// TwinCAT 3 PLC project fms205plc
// ProgramVersion: 3.1.4023.0
// libraries:
//   CmpBitmapPool, * (System)
//   Tc2_Standard, * (Beckhoff Automation GmbH)
//   Tc2_System, * (Beckhoff Automation GmbH)
//   Tc3_Module, * (Beckhoff Automation GmbH)
//   VisuDialogs, * (System)
//   VisuSymbols,3.5.10.0,System
// project tree:
//   / GlobalTextList.TcGTLO, PlcTask.TcTTO (not stored), Visualization Manager.TcVMO (not stored)
//   L1 Architecture/ L1_ModuleBase.TcPOU, L1_Actuator.TcPOU, L1_ControllerBase_SFC.TcPOU, L1_Director.TcPOU, L1_GEMMA.TcDUT, L1_Sensor.TcPOU
//   L2 Module Controllers/ L2_Alimentador_SFC.TcPOU, L2_Cinta_SFC.TcPOU, L2_Evacuador_SFC.TcPOU, L2_MedidorTapa_SFC.TcPOU, L2_PickAndPlace_SFC.TcPOU, L2_PlatoDivisor_SFC.TcPOU, L2_Simple_SFC.TcPOU
//   L3 Modules/ L3_Alimentador.TcPOU, L3_CaptadorInductivo.TcPOU, L3_Cinta.TcPOU, L3_DetectorFotoelectrico.TcPOU, L3_Evacuador.TcPOU, L3_MedidorTapa.TcPOU, L3_PickAndPlace.TcPOU, L3_PlatoDivisor.TcPOU
//   L4 Station Controllers/ L4_FMS205_F1Producir_SFC.TcPOU, L4_FMS205_F2SeqPrep_SFC.TcPOU, L4_FMS205_F3SeqFin_SFC.TcPOU, L4_FMS205_F6Prueba_SFC.TcPOU
//   L5 Station User Interfaces/ L5_Constantes.TcGVL, L5_Panel.TcPOU, L5_FMS205VISU.TcVIS, L5_ImagePool.TcIPO (not stored)
//   L6 Station/ L6_FMS205.TcPOU, L6_Tapas.TcPOU, MAIN.TcPOU
// real-time tasks:
//   TASK PlcTask: cycle T#10ms, priority 20, ADS port 350
// I/O:
//   DEVICE Dispositivo 1 (EtherCAT) (disabled), AmsNetId 192.168.1.58.2.1
//     Terminal 1 (EK1200) [EK1200-5000 EtherCAT Power supply (2A E-Bus)]
//       Terminal 2 (EL1008) [EL1008 8Ch. Dig. Input 24V, 3ms]
//       Terminal 3 (EL1008) [EL1008 8Ch. Dig. Input 24V, 3ms]
//       Terminal 4 (EL2008) [EL2008 8Ch. Dig. Output 24V, 0.5A]
//       Terminal 5 (EL2008) [EL2008 8Ch. Dig. Output 24V, 0.5A]
//       Terminal 6 (EL1008) [EL1008 8Ch. Dig. Input 24V, 3ms]
//       Terminal 7 (EL1008) [EL1008 8Ch. Dig. Input 24V, 3ms]
//       Terminal 8 (EL2008) [EL2008 8Ch. Dig. Output 24V, 0.5A]
//       Terminal 9 (EL2008) [EL2008 8Ch. Dig. Output 24V, 0.5A]
//       Terminal 10 (EL5151) [EL5151 1Ch. Inc. Encoder]
//       Terminal 11 (EL9011) [EL9011 End Terminal]
// variable links:
//   fms205plc/fms205plc Instance <-> Device 1 (EtherCAT)/Term 1 (EK1200)/Term 10 (EL5151)
//     PlcTask Inputs/MAIN.fbFMS205.mdMedidorTapa.dh <-> ENC Inputs/dh
//   fms205plc/fms205plc Instance <-> Device 1 (EtherCAT)/Term 1 (EK1200)/Term 2 (EL1008)
//     PlcTask Inputs/MAIN.fbFMS205.fbPanel.hwPE_Seta <-> Channel 1/PE
//     PlcTask Inputs/MAIN.fbFMS205.fbPanel.hwPM_PulsadorMarcha <-> Channel 3/PM
//     PlcTask Inputs/MAIN.fbFMS205.fbPanel.hwPOC_PulsadorReset <-> Channel 5/POC
//     PlcTask Inputs/MAIN.fbFMS205.fbPanel.hwPS_PulsadorStop <-> Channel 4/PS
//     PlcTask Inputs/MAIN.fbFMS205.fbPanel.hwSM_SelecAutoManual <-> Channel 2/SM
//     PlcTask Inputs/MAIN.fbFMS205.mdCinta.cp0.hwValue <-> Channel 7/cp0
//     PlcTask Inputs/MAIN.fbFMS205.mdCinta.cp1.hwValue <-> Channel 8/cp1
//     PlcTask Inputs/MAIN.fbFMS205.mdCinta.pp.hwValue <-> Channel 6/pp
//   fms205plc/fms205plc Instance <-> Device 1 (EtherCAT)/Term 1 (EK1200)/Term 3 (EL1008)
//     PlcTask Inputs/MAIN.fbFMS205.mdCinta.cp2.hwValue <-> Channel 1/cp2
//   fms205plc/fms205plc Instance <-> Device 1 (EtherCAT)/Term 1 (EK1200)/Term 4 (EL2008)
//     PlcTask Outputs/MAIN.fbFMS205.fbPanel.hwLA_LamparaAlarma <-> Channel 2/LA
//     PlcTask Outputs/MAIN.fbFMS205.fbPanel.hwLM_LamparaMarcha <-> Channel 3/LM
//     PlcTask Outputs/MAIN.fbFMS205.mdAlimentador.FM.hwValue <-> Channel 4/FM
//     PlcTask Outputs/MAIN.fbFMS205.mdCinta.REV.hwValue <-> Channel 6/REV
//     PlcTask Outputs/MAIN.fbFMS205.mdCinta.RUN.hwValue <-> Channel 5/RUN
//     PlcTask Outputs/MAIN.fbFMS205.mdCinta.R_1.hwValue <-> Channel 7/R+
//     PlcTask Outputs/MAIN.fbFMS205.mdCinta.S_1.hwValue <-> Channel 8/S+
//   fms205plc/fms205plc Instance <-> Device 1 (EtherCAT)/Term 1 (EK1200)/Term 5 (EL2008)
//     PlcTask Outputs/MAIN.fbFMS205.fbPanel.hwAS_AvisadorSonoro <-> Channel 1/AS
//   fms205plc/fms205plc Instance <-> Device 1 (EtherCAT)/Term 1 (EK1200)/Term 6 (EL1008)
//     PlcTask Inputs/MAIN.fbFMS205.mdEvacuador.f0.hwValue <-> Channel 6/f0
//     PlcTask Inputs/MAIN.fbFMS205.mdEvacuador.f1.hwValue <-> Channel 7/f1
//     PlcTask Inputs/MAIN.fbFMS205.mdEvacuador.g0.hwValue <-> Channel 8/g0
//     PlcTask Inputs/MAIN.fbFMS205.mdPickAndPlaceCarga.h0.hwValue <-> Channel 1/a0
//     PlcTask Inputs/MAIN.fbFMS205.mdPickAndPlaceCarga.h1.hwValue <-> Channel 2/a1
//     PlcTask Inputs/MAIN.fbFMS205.mdPickAndPlaceCarga.v0.hwValue <-> Channel 3/b0
//     PlcTask Inputs/MAIN.fbFMS205.mdPickAndPlaceCarga.v1.hwValue <-> Channel 4/b1
//     PlcTask Inputs/MAIN.fbFMS205.mdPlatoDivisor.d0.hwValue <-> Channel 5/d0
//   fms205plc/fms205plc Instance <-> Device 1 (EtherCAT)/Term 1 (EK1200)/Term 7 (EL1008)
//     PlcTask Inputs/MAIN.fbFMS205.mdAlimentador.k1.hwValue <-> Channel 6/k1
//     PlcTask Inputs/MAIN.fbFMS205.mdCaptadorInductivo.di.hwValue <-> Channel 7/di
//     PlcTask Inputs/MAIN.fbFMS205.mdDetectorFotoelectrico.df.hwValue <-> Channel 8/df
//     PlcTask Inputs/MAIN.fbFMS205.mdEvacuador.v1.hwValue <-> Channel 1/v1
//     PlcTask Inputs/MAIN.fbFMS205.mdPickAndPlaceDescarga.h0.hwValue <-> Channel 2/h0
//     PlcTask Inputs/MAIN.fbFMS205.mdPickAndPlaceDescarga.h1.hwValue <-> Channel 3/h1
//     PlcTask Inputs/MAIN.fbFMS205.mdPickAndPlaceDescarga.v0.hwValue <-> Channel 4/i0
//     PlcTask Inputs/MAIN.fbFMS205.mdPickAndPlaceDescarga.v1.hwValue <-> Channel 5/i1
//   fms205plc/fms205plc Instance <-> Device 1 (EtherCAT)/Term 1 (EK1200)/Term 8 (EL2008)
//     PlcTask Outputs/MAIN.fbFMS205.mdEvacuador.F_0.hwValue <-> Channel 7/F-
//     PlcTask Outputs/MAIN.fbFMS205.mdEvacuador.F_1.hwValue <-> Channel 6/F+
//     PlcTask Outputs/MAIN.fbFMS205.mdEvacuador.G_1.hwValue <-> Channel 8/G+
//     PlcTask Outputs/MAIN.fbFMS205.mdPickAndPlaceCarga.HOR.hwValue <-> Channel 1/A+
//     PlcTask Outputs/MAIN.fbFMS205.mdPickAndPlaceCarga.PIN.hwValue <-> Channel 3/C+
//     PlcTask Outputs/MAIN.fbFMS205.mdPickAndPlaceCarga.VER.hwValue <-> Channel 2/B+
//     PlcTask Outputs/MAIN.fbFMS205.mdPlatoDivisor.D_1.hwValue <-> Channel 4/D+
//     PlcTask Outputs/MAIN.fbFMS205.mdPlatoDivisor.E_1.hwValue <-> Channel 5/E+
//   fms205plc/fms205plc Instance <-> Device 1 (EtherCAT)/Term 1 (EK1200)/Term 9 (EL2008)
//     PlcTask Outputs/MAIN.fbFMS205.mdAlimentador.K_1.hwValue <-> Channel 5/K+
//     PlcTask Outputs/MAIN.fbFMS205.mdEvacuador.V_1.hwValue <-> Channel 1/V+
//     PlcTask Outputs/MAIN.fbFMS205.mdMedidorTapa.L_1.hwValue <-> Channel 6/L+
//     PlcTask Outputs/MAIN.fbFMS205.mdPickAndPlaceDescarga.HOR.hwValue <-> Channel 2/H+
//     PlcTask Outputs/MAIN.fbFMS205.mdPickAndPlaceDescarga.PIN.hwValue <-> Channel 4/J+
//     PlcTask Outputs/MAIN.fbFMS205.mdPickAndPlaceDescarga.VER.hwValue <-> Channel 3/I+

// ---- L1 Architecture/L1_GEMMA.TcDUT
{attribute 'qualified_only'}
{attribute 'strict'}
TYPE L1_GEMMA :
(
	  (* Modos de la Guia de Estudio de los Modos de Marcha y Parada *)
    (* [Modes du Guide d'Etude des Modes de Marche et d'Arrêt] *)
    (* [Modes of Study Guide of the Modes of Operating and Stopping] *)

    (* Procedimientos de parada [les procédures d'arrets/stop procedures] *)
    A1ParadaInicial, (*  0: parada en el estado inicial
               [arrêt dans etat initial] 
               [stopped in the initial state] *)
    A2ParaFinCiclo, (*  1: parada solicitada a final de ciclo
               [arret demandé en fin de cycle] 
               [requested end cycle stop] *)
    A3ParadaEstado, (*  2: parada solicitada en un estado determinado
               [arret demande dans etat determine] 
               [requested particular state stop] *)
    A4ParadaObtenida, (*  3: parada obtenida
               [arret obtenu] 
               [obteined stop] *)
    A5PreparandoTrasFallo, (*  4: preparacion para la recuperacion del fallo
               [preparation pour remise en route apres defaillance] 
               [preparation for the recovery of the failure] *)
    A6Inicializando, (*  5: situando la PO en el estado inicial
               [mise PO dans état initial] 
               [set the PO in initial state] *)
    A7SituandoEstado, (*  6: situando la PO en un estado determinado
               [mise PO dans état déterminé]
               [set the PO in a certain state] *)

    (* Procedimientos de funcionamiento [les procédures de fonctionnement/operating procedures] *)
    F1ProduccionNormal, (*  7: produccion normal
               [production normale] 
               [normal operation] *)
    F2SecuenciaPreparacion, (*  8: secuencia de preparacion
               [marche de preparation] 
               [preparation sequence] *)
    F3SecuenciaFinalizacion, (*  9: secuencia de finalizacion
               [marche de cloture] 
               [ending sequence] *)
    F4VerificacionSinOrden, (* 10: verificacion en desorden
               [marche de verification dans le desordre] 
               [verification with no order] *)
    F5VerificacionOrdenada, (* 11: verificacion en orden
               [marche de verification dans l'ordre] 
               [verification whit order] *)
    F6Probando, (* 12: prueba
               [marche de test] 
               [test] *)

    (* Procedimientos de fallo [les procédures en défaillances] *)
    D1ParadaEmergencia, (* 13: parada de emergencia
               [arret d'urgence] 
               [emergency stop] *)
    D2TratamientoFallos, (* 14: diagnostico y/o tratamiento de los fallos
               [diagnostic et/ou traitement de la défaillance] 
               [diagnosis and/or treatment of failures] *)
    D3ProducirConFallos  (* 15: produccion a pesar de los fallos
               [production tout de même] 
               [production despite the failures] *)
);
END_TYPE

// ---- L5 Station User Interfaces/L5_Constantes.TcGVL
// {attribute 'qualified_only'}
VAR_GLOBAL CONSTANT
	clModeAFill : DWORD := 16#FF808080;;
	clModeFFill : DWORD := 16#FFFF0000;
	clModeDFill : DWORD := 16#FF800000;
	
	colDesFill		 : DWORD :=16#FFFF0000;	
	colDesFont		 : DWORD :=16#FFFFFFFF;	
	colDesFrameSin	 : DWORD :=16#FFFF0000;		
	colVacFill		 : DWORD :=16#FFF2F2F2;	
	colVacFont		 : DWORD :=16#FF000000;	
	colVacFrameSin	 : DWORD :=16#FFF2F2F2;		
	colTapFill		 : DWORD :=16#FFFFFF00;	
	colTapFont		 : DWORD :=16#FF000000;	
	colTapFrameSin	 : DWORD :=16#FF000000;		
	colClaFill		 : DWORD :=16#FFFFFF00;	
	colClaFont		 : DWORD :=16#FF000000;	
	colClaFrameSin	 : DWORD :=16#FF000000;		
	colOscFill		 : DWORD :=16#FFFFFF00;	
	colOscFont		 : DWORD :=16#FF000000;	
	colOscFrameSin	 : DWORD :=16#FF000000;		
	colAluFill		 : DWORD :=16#FF808080;	
	colAluFont		 : DWORD :=16#FFFFFFFF;	
	colAluFrameSin	 : DWORD :=16#FF000000;	
	colAluFrameOk	 : DWORD :=16#FF00B050;	
	colAluFrameKo	 : DWORD :=16#FFFF0000;
	colBlnFill		 : DWORD :=16#FFFFFFFF;	
	colBlnFont		 : DWORD :=16#FF000000;	
	colBlnFrameSin	 : DWORD :=16#FF000000;	
	colBlnFrameOk	 : DWORD :=16#FF00B050;	
	colBlnFrameKo	 : DWORD :=16#FFFF0000;
	colNgrFill		 : DWORD :=16#FF0D0D0D;	
	colNgrFont		 : DWORD :=16#FFFFFFFF;	
	colNgrFrameSin	 : DWORD :=16#FF000000;	
	colNgrFrameOk	 : DWORD :=16#FF00B050;	
	colNgrFrameKo	 : DWORD :=16#FFFF0000;
	colErrFill		 : DWORD :=16#FFFF0000;	
	colErrFont		 : DWORD :=16#FFFFFFFF;	
	colErrFrameSin	 : DWORD :=16#FF000000;		

	// aparte el grosor de la línea debe establecerse a 3
	colModFillExec	 : DWORD :=16#50FFFF00; // amarillo
	colModFramExec	 : DWORD :=16#FFFFA500; // naranja
	colModFillDone	 : DWORD :=16#5000C000; // verde
	colModFramDone	 : DWORD :=16#FF004000; // verde oscuro
	colModFillReady	 : DWORD :=16#00FFFF00; // amarillo transparente
	colModFramReady	 : DWORD :=16#00FFA500; // naranja transparente
	
	// Posiciones
	MoverMax		: REAL := -1.0;
	MaxAlimeY		: REAL := 100;
	MaxCargaX		: REAL := 80;
	MaxDescaY		: REAL := 90;
	MinCintaX		: REAL := -200;
	MaxCintaX		: REAL := 145;
	
	MaxPosDesca		: REAL := 100;	// mismo valor que deja el brazo de descarga	
	MaxPosEvacu		: REAL := 100;
	MinPosCarro		: REAL := -200;
	MaxPosCarro		: REAL := 145;


END_VAR

// ---- L1 Architecture/L1_ModuleBase.TcPOU
FUNCTION_BLOCK L1_ModuleBase

VAR_INPUT
	dr		: REFERENCE TO L1_Director;
	ID		: BYTE; 		// identificador de la unidad funcional (el módulo)
	Name	: STRING;		// Nombre del módulo (para erroers)
	Execute	: BOOL;
	Ack		: BOOL;
END_VAR

VAR_OUTPUT
	IC			: BOOL;
	Ready		: BOOL;
	Failure		: BOOL;
	FailName 	: STRING;
	Done		: BOOL;
END_VAR

END_FUNCTION_BLOCK

// ---- L1 Architecture/L1_Director.TcPOU
FUNCTION_BLOCK L1_Director
(*

Módulo L1_Director

Entrada: consignas generadas a partir del panel físico, la interfaz de usuario y el estado de la estación
Salida: nuevo estado de Gemma

1. Consignas

	cnA2_FinCiclo:			Solicitud de que la estación se detenga cuando acabe el ciclo
	cnA3_Estado:			Solicitud de que la estación se detenga lo antes posible
	cnA6_Inicializar: 		Solicitud de inicialización de la estación
	
	cnF0_Empezar: 			Solicitud de empezar a Producir/Pobar o continuar después de una parada/fallo
	cnF1_Producir:			Solicitud de producción, incluyendo secuencias de preparación=F2/finalización=F3
	cnF2_Preparar:			Solicitud de que la estación ejecute la secuencia de praparación antes de empezar el lote
	cnF3_Finalizar:			Solicitud de que se ejecute la secuencia de finalización después de acabar el lote
	cnF4_Planta:			Solicitud de paso al modo manual
	cnF5_Funcion:			Solicitud de prueba de grafcets a nivel de módulo
	cnF6_Probar				Solicitud de prueba secuencial de la estación (monolítico)

	cnD1_Emergencia: 		Solicitud de parada de emergencia


2. Estado de la estación

	IC:						La estación cumple las condiciones iniciales
	Failure:				Alguno de los módulos de la estación ha fallado
	EndCycle:				La estación ha terminado un ciclo de producción
	EndBatch:				La estación ha terminado de producir el lote
	IsPaused:				Todos los módulos de la estación se han detenido

3. Modos GEMMA
	A1ParadaInicial:		La estación está parada esperando instrucciones
	A2ParaFinCiclo:			Estación produciendo pero se detendrá cuando se termine el ciclo actual
	A3ParadaEstado:			Estación en marcha pero se detendrá en cuanto alcance un estado estable (IsSafe)
	A4ParadaObtenida: 		La estación está detenida después de alcanzar un estado estable
	A5PreparandoTrasFallo:	La estación está cambiando al modo anterior a que se produjera el fallo
	A6Inicializadndo:		Estación inicializando esperando a que se cumplan las condiciones iniciales
	A7SituandoEstado:		Modo no tratado 
	
	F1ProduccionNormal:		Estación produciendo el lote piezas
	F2SecuenciaPreparacion:	Estación preparándose para producir (evaluando qué hay en cada sector del plato)
	F3SecuenciaFinalizacion:Estación finalizando la producción (vaciando las tapas que quedan en el plato)	
	F4VerificacionSinOrden:	Estación en modo manual
	F5VerificacionOrdenada: Estación ejecutando un Grafcet a nivel de módulo
	F6Probando:				Estación ejecutando el Grafcet secuencial (monolítico)

	D1ParadaEmergencia: 	Estación ha entrado en parada de emergencia
	D2TratamientoFallos:	Estación detenida (o en modo F4) para corregir el fallo que se ha producido
	D3ProducirConFallos:	Estado no tratado

	
*)

VAR CONSTANT
	gmColorArret 	: DWORD := 16#FF808080;
	gmColorFonct 	: DWORD := 16#FF000080;
	gmColorDefail 	: DWORD := 16#FF800000;
END_VAR

VAR_INPUT
	IC 				: BOOL := TRUE; 			// todos los módulos están en condiciones iniciales
	IsPaused		: BOOL := TRUE; 			// estación en estado estable con todos los módulos detenidos
	EndCycle		: BOOL := FALSE;			// se ha completado un ciclo con/sin rechazo/descarga
	EndBatch		: BOOL := FALSE; 			// se han completado todas las tapas del lote
	Failure			: BOOL := FALSE;			// hay al menos un módulo que ha fallado

	cnA1_ParadaIni	: BOOL;
	cnF0_Empezar	: BOOL;
	
	
	cnF1_Producir	: BOOL;
	cnF2_Preparar	: BOOL;
	//IsPrepared		: BOOL := TRUE; 			// secuencia de preparación completada
	
	cnA2_FinCiclo	: BOOL;
	cnA3_Estado		: BOOL;
	cnF3_Finalizar	: BOOL;
	//IsFinished		: BOOL := TRUE; 			// secuencia de finalización completada
	
	cnF5_Funcion	: BOOL; 					// modo verificación ordenada
	cnF6_Probar		: BOOL;

	cnF4_Planta		: BOOL; 					// modo verificación sin orden	
	cnD1_Emergencia	: BOOL; 					// pulsar la seta
	cnA6_Inicializar: BOOL;
	//cnF1_Reanudar	: BOOL;

END_VAR

VAR_OUTPUT
	gmLocalHost		: BOOL 		:= FALSE; 		// TODO - SUSTITUIR ESTO POR LA CONDICIÓN DE LOCALHOST		
	gmModeActual	: L1_GEMMA 	:= L1_GEMMA.A6Inicializando; 		// Modo GEMMA actual
	gmModePrev		: L1_GEMMA; 				// Modo GEMMA anterior al actual
	gmModeColor		: DWORD 	:= gmColorArret;
	Tic				: BOOL		:= FALSE; 		// Se activa y desactiva cada 500 ms
	Clock			: TON;						// Temporizador para activar/desactivar Tic
END_VAR	

VAR
	gmFamiArret		: BOOL 		:= TRUE; 		// Familia de parada
	gmFamiFonct		: BOOL 		:= FALSE; 		// Familia de funcionamiento
	gmFamiDefail	: BOOL 		:= FALSE; 		// Familia de salida de fallos
	
	Speed			: REAL := 100.0;			// Velocidad variable de los controladores
	LastSpeed		: real := 0;			// para calcular sólo si hay cambio de velocidad
	
	
	//---------------------------------- dt_ Defalut Times	
	dt_MaximoTiempoRespuesta	: TIME := T#5S;				// Tiempos generales
	dt_TiempoReinicio			: TIME := T#5S;	
	dt_K_1 						: TIME := T#1S;				// Temporizador empujador tapa
	dt_R_1						: TIME := T#0.5S;			// Temporizador retenedor de la cinta
	dt_S_1						: TIME := T#0.5S;			// Temporizador separador de la cinta
	dt_EP						: TIME := T#0.5S;			// Tiempo de entrada del pale
	dt_TP						: TIME := T#1S;				// Tiempo de transferencia del pale
	dt_XP						: TIME := T#1S;				// Tiempo de salida del pale
	dt_SOL 						: TIME := T#100MS; 			// tiempo después de soltar y antes de subir
	dt_V_1						: TIME := T#5S;				// tiempo máximo succionando sin que se active el sensor v1
	dt_L_1						: TIME := T#1S;				// tiempo máximo de bajada del medidor de tapas
	dt_PIN 						: TIME := T#1S;				// tiempo para pinzar una tapa antes de subir el brazo
	dt_E_1						: TIME := T#400MS;			// tiempo para que el retenedor bloquee el plato
	dt_D_1 						: TIME := T#1.4S;			// tiempo para girar el plato a la siguiente posición
END_VAR


VAR_OUTPUT
	tmMaximoTiempoRespuesta		: TIME := dt_MaximoTiempoRespuesta;
	tmTiempoReinicio			: TIME := dt_TiempoReinicio;	
	tmK_1 						: TIME := dt_K_1;			// Temporizador empujador tapa
	tmR_1						: TIME := dt_R_1;			// Temporizador retenedor de la cinta
	tmS_1						: TIME := dt_S_1;			// Temporizador separador de la cinta
	tmEP						: TIME := dt_EP;			// Tiempo de entrada del pale
	tmTP						: TIME := dt_TP;			// Tiempo de transferencia del pale
	tmXP						: TIME := dt_XP;			// Tiempo de salida del pale
	tmSOL 						: TIME := dt_SOL; 			// tiempo después de soltar y antes de subir
	tmV_1						: TIME := dt_V_1;			// tiempo máximo succionando sin que se active el sensor v1
	tmL_1						: TIME := dt_L_1;		// tiempo máximo de bajada del medidor de tapas
	tmPIN 						: TIME := dt_PIN;		// tiempo para pinzar una tapa antes de subir el brazo
	tmE_1						: TIME := dt_E_1;		// tiempo para que el retenedor bloquee el plato
	tmD_1 						: TIME := dt_D_1;		// tiempo para girar el plato a la siguiente posición
END_VAR

METHOD ProcessCycle : BOOL
// Actualiza el reloj y la veloidad cada medio segundo
Clock(IN := NOT Clock.Q, PT:=T#500MS);
IF Clock.Q THEN
	Tic := NOT Tic;
	UpdateSpeed();
END_IF


IF cnD1_Emergencia AND NOT cnF4_Planta THEN
    gmModeActual 		:= L1_GEMMA.D1ParadaEmergencia;
//	gmModePrev 			:= L1_GEMMA.D1ParadaEmergencia;
//	IF cnF4_Planta THEN 				
//		gmModePrev := L1_GEMMA.D1ParadaEmergencia
//		gmModeActual := L1_GEMMA.F4VerificacionSinOrden;
//	ELSE
//		; // desde emergencia se puede pasar a F4 (desarmando la seta)				
//	END_IF
//		
	
ELSIF cnA6_Inicializar and not cnF4_Planta THEN 
    gmModeActual 		:= L1_GEMMA.A6Inicializando;
	// gmModePrev 			:= L1_GEMMA.L1_GEMMA.A6Inicializando;	

END_IF
	
    CASE gmModeActual OF
		
	
        (* ------------------------------------------------------------ Procedimientos de parada *)
		
        L1_GEMMA.A6Inicializando: (* A6 -> A1 o F4 *)
			gmModePrev := L1_GEMMA.A6Inicializando;
            IF IC THEN 
                gmModeActual := L1_GEMMA.A1ParadaInicial;
			ELSIF cnF4_Planta THEN 				
                gmModeActual := L1_GEMMA.F4VerificacionSinOrden;
            END_IF

			
			
			
        L1_GEMMA.A1ParadaInicial: (* A1 -> A6, F4, F5, F2 o F6 *)
			gmModePrev := L1_GEMMA.A1ParadaInicial;
            IF NOT IC THEN // IF NOT Restaurada THEN
                gmModeActual := L1_GEMMA.A6Inicializando;				
            ELSIF cnF4_Planta THEN 				
                gmModeActual := L1_GEMMA.F4VerificacionSinOrden;				
			ELSIF cnF5_Funcion THEN 
				gmModeActual := L1_GEMMA.F5VerificacionOrdenada;             
			ELSIF cnF1_Producir AND cnF0_Empezar THEN
                gmModeActual := L1_GEMMA.F2SecuenciaPreparacion;
			ELSIF cnF6_Probar AND cnF0_Empezar THEN
				gmModeActual := L1_GEMMA.F6Probando;
			ELSE
				; // Esperar a que se pulse el bortón de marcha
            END_IF

			
			
        L1_GEMMA.F4VerificacionSinOrden: (* F4 -> ModePrev *)
            //IF Failure THEN
			//	gmModeActual := L1_GEMMA.D2TratamientoFallos;				
            //ELSIF NOT cnF4_Planta THEN
			IF NOT cnF4_Planta THEN 				
				gmModeActual := gmModePrev; // al salir del modo planta volver al modo previo				
            ELSE                
                ; // Seguir en modo manual
            END_IF

			
			
		L1_GEMMA.F1ProduccionNormal, 		
        L1_GEMMA.A2ParaFinCiclo,
        L1_GEMMA.F2SecuenciaPreparacion, 	
		L1_GEMMA.F3SecuenciaFinalizacion, 	
        L1_GEMMA.F5VerificacionOrdenada,  	
		L1_GEMMA.F6Probando: 				        
			// retorno desde tratamiento de errores y planta
			IF gmModeActual=L1_GEMMA.F5VerificacionOrdenada THEN
				gmModePrev := L1_GEMMA.A1ParadaInicial; 								// F5 retorna a A1
			ELSE
				gmModePrev := gmModeActual;												// Resto retorna donde quedó			
			END_IF			
			
			// cambios de modo actual
            IF Failure THEN 															// cualquiera -> D2
                gmModeActual := L1_GEMMA.D2TratamientoFallos;
            ELSIF cnA3_Estado THEN				
				gmModeActual := L1_GEMMA.A3ParadaEstado; 								// cualquiera -> A3
			ELSIF cnF4_Planta THEN 				
                gmModeActual := L1_GEMMA.F4VerificacionSinOrden;						// cualquiera -> F4
            ELSIF gmModeActual=L1_GEMMA.F2SecuenciaPreparacion AND NOT cnF2_Preparar THEN 	// F2-> F1
                gmModeActual:= L1_GEMMA.F1ProduccionNormal;
			ELSIF gmModeActual=L1_GEMMA.F1ProduccionNormal AND cnA2_FinCiclo THEN 		// F1 -> A2				
				gmModeActual:= L1_GEMMA.A2ParaFinCiclo;
			ELSIF gmModeActual=L1_GEMMA.A2ParaFinCiclo AND EndCycle THEN 				// A2 -> A3
				gmModePrev  := L1_GEMMA.F1ProduccionNormal; 							// A2 -> A3 ... -> F1
                gmModeActual:= L1_GEMMA.A3ParadaEstado;
			ELSIF gmModeActual=L1_GEMMA.F1ProduccionNormal AND EndBatch THEN 			// F1-> F3
                gmModeActual:= L1_GEMMA.F3SecuenciaFinalizacion;
			ELSIF gmModeActual=L1_GEMMA.F3SecuenciaFinalizacion AND NOT cnF3_Finalizar THEN // F3 -> A1
				gmModeActual:= L1_GEMMA.A1ParadaInicial;
			ELSIF gmModeActual=L1_GEMMA.F5VerificacionOrdenada AND NOT cnF5_Funcion THEN // F5 -> A1
				gmModeActual:= L1_GEMMA.A1ParadaInicial;				
			ELSIF gmModeActual=L1_GEMMA.F6Probando AND NOT cnF6_Probar THEN 			// F6 -> A1
				gmModeActual:= L1_GEMMA.A1ParadaInicial; 
            ELSE                
                ; // continuar con la preparación/producción/finalización
            END_IF
			

			
        L1_GEMMA.A3ParadaEstado: 
			IF Failure THEN																// A3 -> D2
                gmModeActual := L1_GEMMA.D2TratamientoFallos;
			ELSIF IsPaused THEN															// A3 -> A4
                gmModeActual := L1_GEMMA.A4ParadaObtenida;
            ELSE
                ; // Seguir produciendo hasta que todos los módulos paren en un estado estable
            END_IF
            			
        L1_GEMMA.A4ParadaObtenida:
			IF cnF0_Empezar THEN														// A4 -> retorna
				gmModeActual := gmModePrev; // retomar el estado antes de la parada
			ELSE
				; // seguir parada hasta la consigna de reanudar	
			END_IF
                    
		L1_GEMMA.A5PreparandoTrasFallo:
			gmModeActual := gmModePrev;		// Volver al estado anterior al fallo 
			
        L1_GEMMA.A7SituandoEstado: (* Situando la PO en un estado determinado *)
            ; // estado no tratado en la FMS205

			
			
        (* ------------------------------------------------------------ Procedimientos de funcionamiento *)
        
			
			
			
			
        	
			
        (* ------------------------------------------------------------ Procedimientos de defecto *)
        L1_GEMMA.D1ParadaEmergencia: (* Parada de emergencia *)
			IF NOT cnD1_Emergencia THEN //  TODO CONSIGNA DE EMERGENCIA DEBE TENER ENCUENTA LA POC
                gmModeActual := L1_GEMMA.A6Inicializando; // Al quitar la parada de emergencia hay que reinicializar la estación
			ELSIF cnF4_Planta then							// desde A1 se puede entrar F4 para arreglar el problema
				gmModePrev := L1_GEMMA.D1ParadaEmergencia;
				gmModeActual := L1_GEMMA.F4VerificacionSinOrden;
            ELSE                
                ; // Esperar a que se quite la parada de emergencia
            END_IF
			
        L1_GEMMA.D2TratamientoFallos: (* Diagnostico/tratamiento de los fallos *)
            IF NOT Failure THEN // el fallo se resuelve por sí solo (no debería pasar)
                gmModeActual := L1_GEMMA.A5PreparandoTrasFallo;
			ELSIF cnF4_Planta THEN // se pasa a modo F4 para arreglarlo
				gmModeActual := L1_GEMMA.F4VerificacionSinOrden;
            ELSIF cnF0_Empezar THEN // se pulsa Marcha para intentar recuperar                
                gmModeActual := L1_GEMMA.A5PreparandoTrasFallo;
            END_IF

        L1_GEMMA.D3ProducirConFallos: (* Produccion a pesar de los fallos *)
            ; // estado no tratado en la FMS205

    END_CASE
// END_IF

(* PARAMETROS DE SALIDA *)
gmFamiArret  := (gmModeActual >= L1_GEMMA.A1ParadaInicial) AND (gmModeActual <= L1_GEMMA.A7SituandoEstado);
gmFamiFonct  := (gmModeActual >= L1_GEMMA.F1ProduccionNormal) AND (gmModeActual <= L1_GEMMA.F6Probando);
gmFamiDefail := (gmModeActual >= L1_GEMMA.D1ParadaEmergencia) AND (gmModeActual <= L1_GEMMA.D3ProducirConFallos);
gmModeColor := SEL(gmFamiArret,SEL(gmFamiFonct, gmColorDefail, gmColorFonct), gmColorArret);

UpdateSpeed();
//UpdateUi(pn:=pn);
END_METHOD

METHOD UpdateSpeed : BOOL

VAR
	factor : REAL;
END_VAR
IF Speed <= 0 THEN
	Speed := 1;
ELSIF Speed<>LastSpeed THEN
	LastSpeed := Speed; // sólo se ejecuta el código la primera vez que cambia la velocidad
	
	factor := 100.0/Speed;
	
	tmMaximoTiempoRespuesta		:= TO_TIME(TO_REAL(dt_MaximoTiempoRespuesta) * factor);
	tmTiempoReinicio			:= TO_TIME(TO_REAL(dt_TiempoReinicio) * factor);
	tmK_1 						:= TO_TIME(TO_REAL(dt_K_1) * factor);					// Temporizador empujador tapa
	tmR_1						:= TO_TIME(TO_REAL(dt_R_1) * factor);					// Temporizador retenedor de la cinta
	tmS_1						:= TO_TIME(TO_REAL(dt_S_1) * factor);					// Temporizador separador de la cinta
	tmEP						:= TO_TIME(TO_REAL(dt_EP) * factor);					// Tiempo de entrada del pale
	tmTP						:= TO_TIME(TO_REAL(dt_TP) * factor);					// Tiempo de transferencia del pale
	tmXP						:= TO_TIME(TO_REAL(dt_XP) * factor);					// Tiempo de salida del pale
	tmSOL 						:= TO_TIME(TO_REAL(dt_SOL) * factor); 					// tiempo después de soltar y antes de subir
	tmV_1						:= TO_TIME(TO_REAL(dt_V_1) * factor);					// tiempo máximo succionando sin que se active el sensor v1
	tmL_1						:= TO_TIME(TO_REAL(dt_L_1) * factor);					// tiempo máximo de bajada del medidor de tapas
	tmPIN 						:= TO_TIME(TO_REAL(dt_PIN) * factor);					// tiempo para pinzar una tapa antes de subir el brazo
	tmE_1						:= TO_TIME(TO_REAL(dt_E_1) * factor);					// tiempo para que el retenedor bloquee el plato
	tmD_1 						:= TO_TIME(TO_REAL(dt_D_1) * factor);					// tiempo para girar el plato a la siguiente posición
	
END_IF
END_METHOD

END_FUNCTION_BLOCK

// ---- L1 Architecture/L1_Actuator.TcPOU
FUNCTION_BLOCK L1_Actuator

VAR CONSTANT
END_VAR

VAR_OUTPUT
	uiValue			: BOOL;					// Vinculación a la visualización
	uiToolTip		: STRING;				// Tooltip en la visualización
END_VAR

VAR
	hwValue AT %Q*	: BOOL;					// Vinculación al hardware de la estación	
END_VAR

METHOD ForceValue : BOOL
VAR_INPUT
	NewValue : BOOL;
END_VAR
uiValue := NewValue;
hwValue := NewValue;
END_METHOD

METHOD ProcessCycle : BOOL
VAR_INPUT
	gmMode		: L1_GEMMA;
	sfcValue 	: BOOL;		// estado del actuador devuelto por el Grafcet
END_VAR
IF gmMode = L1_GEMMA.F4VerificacionSinOrden THEN	
	hwValue := uiValue;	// Actualizar el hardware con la entrada desde la visualización
ELSE	
	hwValue := sfcValue; // Actualizar el hardware y la visualicación con la entrada desde el Grafcet
	uiValue := sfcValue;
END_IF
END_METHOD

END_FUNCTION_BLOCK

// ---- L1 Architecture/L1_ControllerBase_SFC.TcPOU
FUNCTION_BLOCK L1_ControllerBase_SFC

VAR_INPUT
	dr			: REFERENCE TO L1_Director;		// acceso a todos los tiempos de espera
	IC			: BOOL;
	Execute		: BOOL;
	Ack			: BOOL;	
	SFCPause	: BOOL;
	SFCReset	: BOOL;
	UnsafeStop 	: BOOL;
	Clocks		: ARRAY[1..MAX_ERRORS]	OF TON; 
END_VAR

VAR_OUTPUT
	Ready		: BOOL;
	Executing	: BOOL;
	_Performed	: BOOL;					// Para poner la primera vez que se leen los sensores o se gira el plato
	Done		: BOOL := FALSE;
	Timed		: ARRAY[1..MAX_ERRORS]	OF BOOL; 
	NumError	: UINT := 0;
	gmModePrev	: L1_GEMMA := L1_GEMMA.A6Inicializando;	
	colPicFill	: DWORD; // color para destacar en la foto según esté Ready (tranparente), Ejecutando (amarillo) o Esperando Ack (verde) 
	colPicFram	: DWORD; // color del marco  	
END_VAR

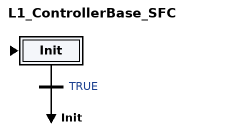
INITIAL_STEP Init:
END_STEP
TRANSITION FROM Init TO Init
    := TRUE;
END_TRANSITION

METHOD FB_init : BOOL

VAR_INPUT
	bInitRetains : BOOL; // if TRUE, the retain variables are initialized (warm start / cold start)
	bInCopyCode : BOOL;  // if TRUE, the instance afterwards gets moved into the copy code (online change)
END_VAR

VAR 
	I: UINT;
END_VAR
NumError		:= 0;					// Inicializar el estado a 0 (no hay error)
_Performed		:= FALSE;
UnsafeStop 		:= FALSE;
Done			:= FALSE;
gmModePrev		:= L1_GEMMA.A6Inicializando;

FOR I:=1 TO MAX_ERRORS DO				// Inicializar todos los flags de etapas temporizadas
	Timed[i] 		:= FALSE;
END_FOR
END_METHOD

METHOD IsPaused : BOOL
IsPaused := SFCPause;
END_METHOD

PROPERTY Performed : BOOL
GET
Performed := _Performed;
END_GET
SET
_Performed := Performed;
END_SET
END_PROPERTY

METHOD ProcessCycle : BOOL

VAR_INPUT
	gmMode : L1_GEMMA;
END_VAR

VAR 
	i : UINT;
END_VAR
// Tratamiento del reset
IF gmModePrev<>gmMode AND gmMode=L1_GEMMA.A6Inicializando THEN
	gmModePrev	:= gmMode;
	SFCReset 	:= TRUE;
	Ready		:= FALSE; 
	Executing	:= FALSE;
	_Performed	:= FALSE;				// Para poner la primera vez que se leen los sensores o se gira el plato
	Done		:= FALSE;
	NumError	:= 0;
	colPicFill	:= colModFillReady;  
	colPicFram	:= colModFramReady;   	
ELSE
	SFCReset 	:= FALSE;
END_IF
gmModePrev := gmMode;

// Tratamiento de la parada
SFCPause := NOT UnsafeStop AND (NumError <> 0 
	OR gmMode=L1_GEMMA.A3ParadaEstado OR gmMode=L1_GEMMA.A4ParadaObtenida or gmMode=L1_GEMMA.D1ParadaEmergencia);

// Tratamiento de errores
FOR i:= 1 TO MAX_ERRORS DO			
	Clocks[i](IN:= Timed[i], PT:=MAX_TIMEOUT);
	IF Clocks[i].Q THEN								// si saltó algún temporizador, devolver su número como error
		NumError := i;
		EXIT;
	END_IF
END_FOR


// Tratamiento del color en la foto
IF Ready THEN
	Executing 	:= FALSE;
	Performed 	:= FALSE;
	colPicFill	:= colModFillReady;
	colPicFram	:= colModFramReady;
ELSIF Done THEN
	Executing 	:= FALSE;
	colPicFill	:= colModFillDone;
	colPicFram	:= colModFramDone;	
ELSE
	Executing 	:= TRUE;
	colPicFill	:= colModFillExec;
	colPicFram	:= colModFramExec;	
END_IF
END_METHOD

METHOD ResetError : BOOL
NumError := 0;
END_METHOD

END_FUNCTION_BLOCK

// ---- L1 Architecture/L1_Sensor.TcPOU
FUNCTION_BLOCK L1_Sensor

VAR_OUTPUT
	uiValue			: BOOL;					
END_VAR

VAR	
	hwValue AT %I*	: BOOL;					// Vinculación al hardware de la estación
	uiToolTip		: STRING;				// Tooltip en la visualización
END_VAR

METHOD ProcessCycle : BOOL
VAR_INPUT
	LocalHost	: BOOL;
END_VAR
VAR_OUTPUT
	sfcValue 	: BOOL;		// estado del sensor que se entregará al Grafcet
END_VAR
IF LocalHost THEN	
	hwValue := uiValue; 	// simulando la estación, el valor del sensor depende de la interfaz	
ELSE	
	uiValue := hwValue; 	// ejecutando en la estación, el valor de la visualización depende del hardware
END_IF
sfcValue := hwValue;		// estado del sensor que se entregará al Grafcet
END_METHOD

END_FUNCTION_BLOCK

// ---- L2 Module Controllers/L2_Alimentador_SFC.TcPOU
FUNCTION_BLOCK L2_Alimentador_SFC EXTENDS L1_ControllerBase_SFC

VAR_INPUT 					// Sensores y comandos
	k1	: BOOL; 			// Sensor de empujador tapa delante
	Alimentar :BOOL;
END_VAR

VAR_OUTPUT					// Actuadores
	Leyendo: BOOL;	
	K_1: BOOL; 				// Actuador de empujador tapa avanza	 
	FM : BOOL; 
END_VAR

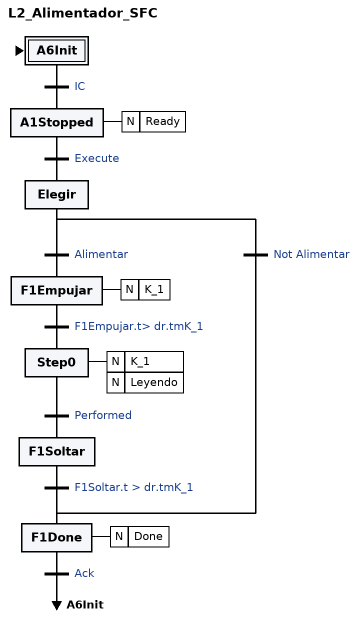
INITIAL_STEP A6Init:
END_STEP
TRANSITION FROM A6Init TO A1Stopped
    := IC;
END_TRANSITION
STEP A1Stopped:
    Ready(N);
END_STEP
TRANSITION FROM A1Stopped TO Elegir
    := Execute;
END_TRANSITION
STEP Elegir:
END_STEP
TRANSITION FROM Elegir TO F1Empujar
    := Alimentar;
END_TRANSITION
STEP F1Empujar:
    K_1(N);
END_STEP
TRANSITION FROM F1Empujar TO Step0
    := F1Empujar.t> dr.tmK_1;
END_TRANSITION
STEP Step0:
    K_1(N);
    Leyendo(N);
END_STEP
TRANSITION FROM Step0 TO F1Soltar
    := Performed;
END_TRANSITION
STEP F1Soltar:
END_STEP
TRANSITION FROM F1Soltar TO F1Done
    := F1Soltar.t > dr.tmK_1;
END_TRANSITION
TRANSITION FROM Elegir TO F1Done
    := Not Alimentar;
END_TRANSITION
STEP F1Done:
    Done(N);
END_STEP
TRANSITION FROM F1Done TO A6Init
    := Ack;
END_TRANSITION

END_FUNCTION_BLOCK

// ---- L2 Module Controllers/L2_Cinta_SFC.TcPOU
FUNCTION_BLOCK L2_Cinta_SFC  EXTENDS L1_ControllerBase_SFC

VAR_INPUT 					// Sensores y comandos
	Situar		: BOOL;
	Transferir	: BOOL;	
	pp			: BOOL; 	// presencia de pale
	cp0			: BOOL;
	cp1			: BOOL;
	cp2			: BOOL;
END_VAR

VAR_OUTPUT					// Actuadores
	RUN			: BOOL; 	// activa motor
	REV			: BOOL; 	// invierte motor
	R_1			: BOOL; 	// retenedor baja
	S_1			: BOOL; 	// separador sube
END_VAR

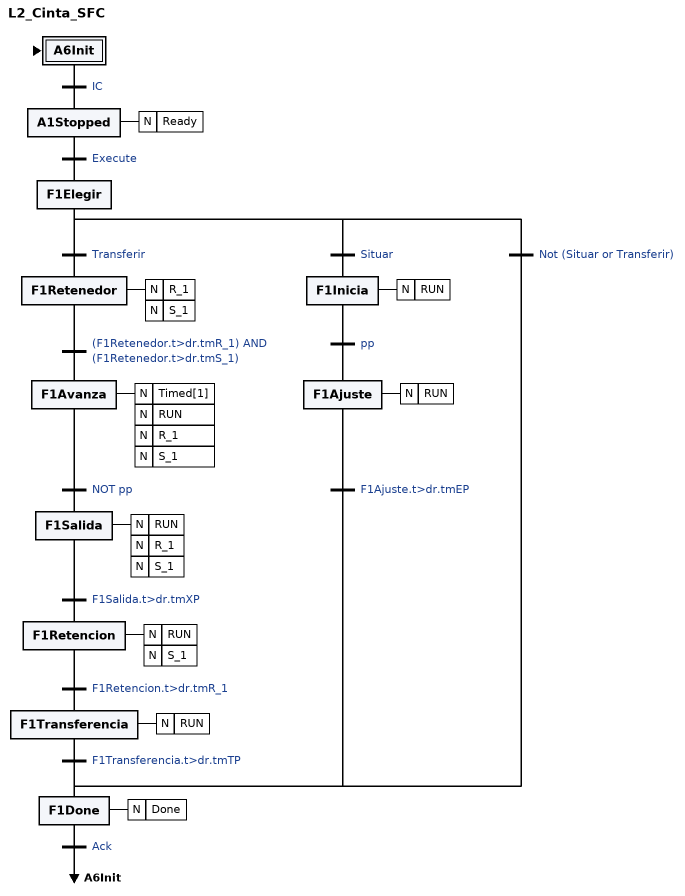
INITIAL_STEP A6Init:
END_STEP
TRANSITION FROM A6Init TO A1Stopped
    := IC;
END_TRANSITION
STEP A1Stopped:
    Ready(N);
END_STEP
TRANSITION FROM A1Stopped TO F1Elegir
    := Execute;
END_TRANSITION
STEP F1Elegir:
END_STEP
TRANSITION FROM F1Elegir TO F1Retenedor
    := Transferir;
END_TRANSITION
STEP F1Retenedor:
    R_1(N);
    S_1(N);
END_STEP
TRANSITION FROM F1Retenedor TO F1Avanza
    := (F1Retenedor.t>dr.tmR_1) AND (F1Retenedor.t>dr.tmS_1);
END_TRANSITION
STEP F1Avanza:
    Timed[1](N);
    RUN(N);
    R_1(N);
    S_1(N);
END_STEP
TRANSITION FROM F1Avanza TO F1Salida
    := NOT pp;
END_TRANSITION
STEP F1Salida:
    RUN(N);
    R_1(N);
    S_1(N);
END_STEP
TRANSITION FROM F1Salida TO F1Retencion
    := F1Salida.t>dr.tmXP;
END_TRANSITION
STEP F1Retencion:
    RUN(N);
    S_1(N);
END_STEP
TRANSITION FROM F1Retencion TO F1Transferencia
    := F1Retencion.t>dr.tmR_1;
END_TRANSITION
STEP F1Transferencia:
    RUN(N);
END_STEP
TRANSITION FROM F1Transferencia TO F1Done
    := F1Transferencia.t>dr.tmTP;
END_TRANSITION
TRANSITION FROM F1Elegir TO F1Inicia
    := Situar;
END_TRANSITION
STEP F1Inicia:
    RUN(N);
END_STEP
TRANSITION FROM F1Inicia TO F1Ajuste
    := pp;
END_TRANSITION
STEP F1Ajuste:
    RUN(N);
END_STEP
TRANSITION FROM F1Ajuste TO F1Done
    := F1Ajuste.t>dr.tmEP;
END_TRANSITION
TRANSITION FROM F1Elegir TO F1Done
    := Not (Situar or Transferir);
END_TRANSITION
STEP F1Done:
    Done(N);
END_STEP
TRANSITION FROM F1Done TO A6Init
    := Ack;
END_TRANSITION

END_FUNCTION_BLOCK

// ---- L2 Module Controllers/L2_Evacuador_SFC.TcPOU
FUNCTION_BLOCK L2_Evacuador_SFC EXTENDS L1_ControllerBase_SFC

VAR_INPUT 				// Sensores y comandos
	Evacuar		: BOOL; // Hay que evacuar la tapa en la posición del módulo
	f0        	: BOOL; (* gh0 (nombre=f0  c=I22 B=J2 b=22 módulo=EL1008 T=6  C=6 etiqueta=-B10, input) Pick and place de rechazo detrás *)
    f1        	: BOOL; (* gh1 (nombre=f1  c=I23 B=J2 b=06 módulo=EL1008 T=6  C=6 etiqueta=-B11, input) Pick and place de rechazo delante *)
    g0        	: BOOL; (* gv1 (nombre=g0  c=I24 B=J2 b=31 módulo=EL1008 T=6  C=6 etiqueta=-B12, input) Pick and place de rechazo arriba *)
    v1        	: BOOL; (* ge1 (nombre=v1  c=I25 B=J1 b=25 módulo=EL1008 T=7  C=7 etiqueta=-B13, input) Pick and place de rechazo vacío *)
END_VAR

VAR_OUTPUT				// Actuadores
	F_1       	: BOOL; (* gHRA (nombre=F+  c=Q22 B=J2  b=35 módulo=EL2008 T=8 C=8 etiqueta=-Y8,  output) Pick and place de rechazo avanza (afuera) *)
    F_0       	: BOOL; (* gHRR (nombre=F-  c=Q23 B=J2  b=32 módulo=EL2008 T=8 C=8 etiqueta=-Y9,  output) Pick and place de rechazo retrocede *)
    G_1       	: BOOL; (* gVER (nombre=G+  c=Q24 B=J2  b=11 módulo=EL2008 T=8 C=8 etiqueta=-Y10, output) Pick and place de rechazo baja *)
    V_1       	: BOOL; (* gEYE (nombre=V+  c=Q25 B=J2  b=08 módulo=EL2008 T=9 C=9 etiqueta=-Y11, output) Pick and place de rechazo succiona *)
END_VAR

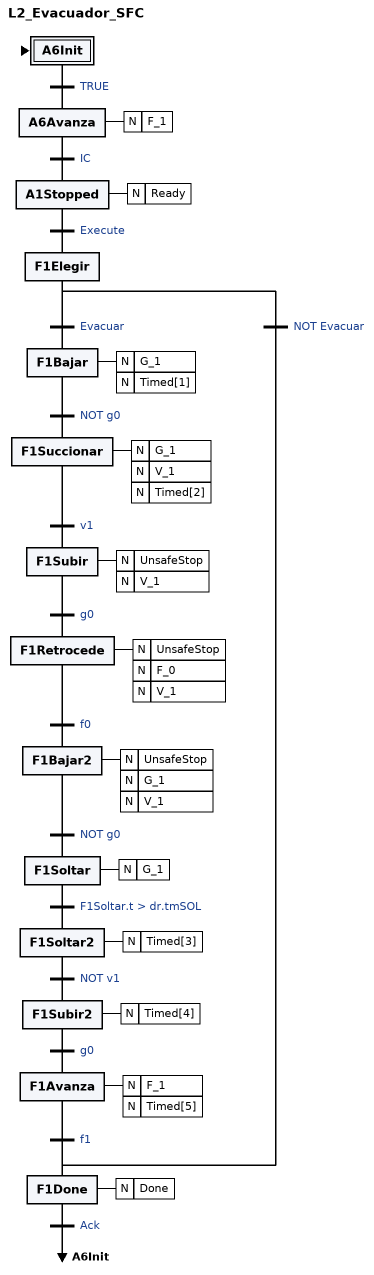
INITIAL_STEP A6Init:
END_STEP
TRANSITION FROM A6Init TO A6Avanza
    := TRUE;
END_TRANSITION
STEP A6Avanza:
    F_1(N);
END_STEP
TRANSITION FROM A6Avanza TO A1Stopped
    := IC;
END_TRANSITION
STEP A1Stopped:
    Ready(N);
END_STEP
TRANSITION FROM A1Stopped TO F1Elegir
    := Execute;
END_TRANSITION
STEP F1Elegir:
END_STEP
TRANSITION FROM F1Elegir TO F1Bajar
    := Evacuar;
END_TRANSITION
STEP F1Bajar:
    G_1(N);
    Timed[1](N);
END_STEP
TRANSITION FROM F1Bajar TO F1Succionar
    := NOT g0;
END_TRANSITION
STEP F1Succionar:
    G_1(N);
    V_1(N);
    Timed[2](N);
END_STEP
TRANSITION FROM F1Succionar TO F1Subir
    := v1;
END_TRANSITION
STEP F1Subir:
    UnsafeStop(N);
    V_1(N);
END_STEP
TRANSITION FROM F1Subir TO F1Retrocede
    := g0;
END_TRANSITION
STEP F1Retrocede:
    UnsafeStop(N);
    F_0(N);
    V_1(N);
END_STEP
TRANSITION FROM F1Retrocede TO F1Bajar2
    := f0;
END_TRANSITION
STEP F1Bajar2:
    UnsafeStop(N);
    G_1(N);
    V_1(N);
END_STEP
TRANSITION FROM F1Bajar2 TO F1Soltar
    := NOT g0;
END_TRANSITION
STEP F1Soltar:
    G_1(N);
END_STEP
TRANSITION FROM F1Soltar TO F1Soltar2
    := F1Soltar.t > dr.tmSOL;
END_TRANSITION
STEP F1Soltar2:
    Timed[3](N);
END_STEP
TRANSITION FROM F1Soltar2 TO F1Subir2
    := NOT v1;
END_TRANSITION
STEP F1Subir2:
    Timed[4](N);
END_STEP
TRANSITION FROM F1Subir2 TO F1Avanza
    := g0;
END_TRANSITION
STEP F1Avanza:
    F_1(N);
    Timed[5](N);
END_STEP
TRANSITION FROM F1Avanza TO F1Done
    := f1;
END_TRANSITION
TRANSITION FROM F1Elegir TO F1Done
    := NOT Evacuar;
END_TRANSITION
STEP F1Done:
    Done(N);
END_STEP
TRANSITION FROM F1Done TO A6Init
    := Ack;
END_TRANSITION

END_FUNCTION_BLOCK

// ---- L2 Module Controllers/L2_MedidorTapa_SFC.TcPOU
FUNCTION_BLOCK L2_MedidorTapa_SFC EXTENDS L1_ControllerBase_SFC

VAR_INPUT 							// Sensores y comandos
	dh					: UINT; 	// Detector valor altura 
	Medir				: BOOL; // Lectura_Registrada	: BOOL;		// La lectura de la altura ha terminado 	
END_VAR

VAR_OUTPUT							// Actuadores
	L_1: BOOL; 						// Medidor de altura baja
	Leyendo: BOOL;
END_VAR

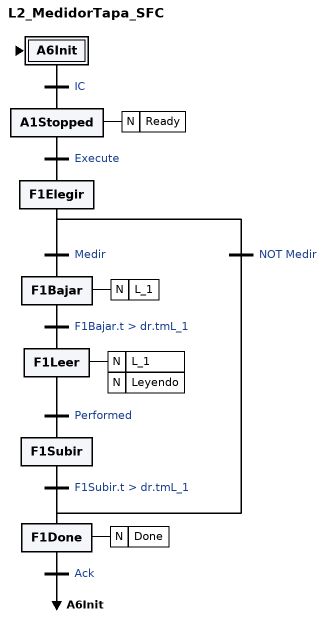
INITIAL_STEP A6Init:
END_STEP
TRANSITION FROM A6Init TO A1Stopped
    := IC;
END_TRANSITION
STEP A1Stopped:
    Ready(N);
END_STEP
TRANSITION FROM A1Stopped TO F1Elegir
    := Execute;
END_TRANSITION
STEP F1Elegir:
END_STEP
TRANSITION FROM F1Elegir TO F1Bajar
    := Medir;
END_TRANSITION
STEP F1Bajar:
    L_1(N);
END_STEP
TRANSITION FROM F1Bajar TO F1Leer
    := F1Bajar.t > dr.tmL_1;
END_TRANSITION
STEP F1Leer:
    L_1(N);
    Leyendo(N);
END_STEP
TRANSITION FROM F1Leer TO F1Subir
    := Performed;
END_TRANSITION
STEP F1Subir:
END_STEP
TRANSITION FROM F1Subir TO F1Done
    := F1Subir.t > dr.tmL_1;
END_TRANSITION
TRANSITION FROM F1Elegir TO F1Done
    := NOT Medir;
END_TRANSITION
STEP F1Done:
    Done(N);
END_STEP
TRANSITION FROM F1Done TO A6Init
    := Ack;
END_TRANSITION

END_FUNCTION_BLOCK

// ---- L2 Module Controllers/L2_PickAndPlace_SFC.TcPOU
FUNCTION_BLOCK L2_PickAndPlace_SFC EXTENDS L1_ControllerBase_SFC

VAR_INPUT 				// Sensores y comandos
	h0		: BOOL; 	(* Final de carrera horizontal retraida *)
	h1		: BOOL; 	(* Final de carrera horizontal extendido *)
	v1		: BOOL; 	(*Final de carrera vertical abajo*)
	v0		: BOOL; 	(*Final de carrera vertical arriba*)
	Mover	: BOOL;
END_VAR

VAR_OUTPUT			// Actuadores
	HOR		: BOOL; (* Actuador de extension de brazo horizontal *)
	VER		: BOOL; (* Actuador de movimiento vertical de brazo*)
	PIN		: BOOL; (*Actuador de pinza de brazo*)
END_VAR

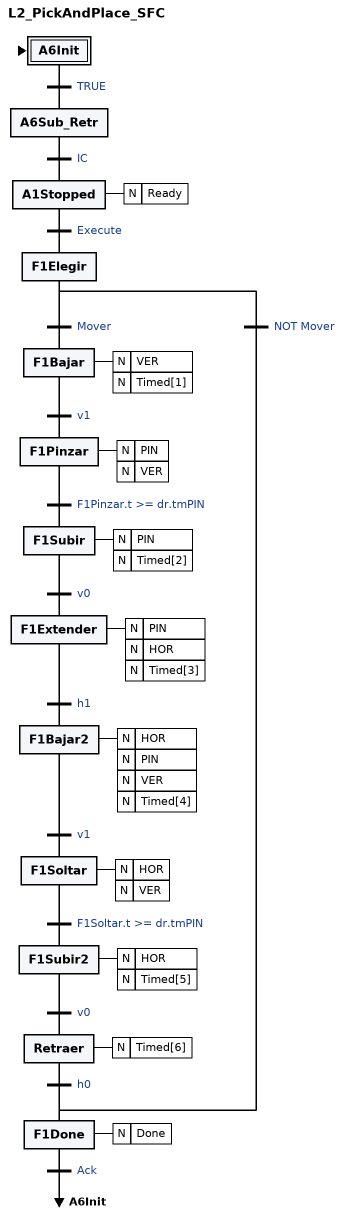
INITIAL_STEP A6Init:
END_STEP
TRANSITION FROM A6Init TO A6Sub_Retr
    := TRUE;
END_TRANSITION
STEP A6Sub_Retr:
END_STEP
TRANSITION FROM A6Sub_Retr TO A1Stopped
    := IC;
END_TRANSITION
STEP A1Stopped:
    Ready(N);
END_STEP
TRANSITION FROM A1Stopped TO F1Elegir
    := Execute;
END_TRANSITION
STEP F1Elegir:
END_STEP
TRANSITION FROM F1Elegir TO F1Bajar
    := Mover;
END_TRANSITION
STEP F1Bajar:
    VER(N);
    Timed[1](N);
END_STEP
TRANSITION FROM F1Bajar TO F1Pinzar
    := v1;
END_TRANSITION
STEP F1Pinzar:
    PIN(N);
    VER(N);
END_STEP
TRANSITION FROM F1Pinzar TO F1Subir
    := F1Pinzar.t >= dr.tmPIN;
END_TRANSITION
STEP F1Subir:
    PIN(N);
    Timed[2](N);
END_STEP
TRANSITION FROM F1Subir TO F1Extender
    := v0;
END_TRANSITION
STEP F1Extender:
    PIN(N);
    HOR(N);
    Timed[3](N);
END_STEP
TRANSITION FROM F1Extender TO F1Bajar2
    := h1;
END_TRANSITION
STEP F1Bajar2:
    HOR(N);
    PIN(N);
    VER(N);
    Timed[4](N);
END_STEP
TRANSITION FROM F1Bajar2 TO F1Soltar
    := v1;
END_TRANSITION
STEP F1Soltar:
    HOR(N);
    VER(N);
END_STEP
TRANSITION FROM F1Soltar TO F1Subir2
    := F1Soltar.t >= dr.tmPIN;
END_TRANSITION
STEP F1Subir2:
    HOR(N);
    Timed[5](N);
END_STEP
TRANSITION FROM F1Subir2 TO Retraer
    := v0;
END_TRANSITION
STEP Retraer:
    Timed[6](N);
END_STEP
TRANSITION FROM Retraer TO F1Done
    := h0;
END_TRANSITION
TRANSITION FROM F1Elegir TO F1Done
    := NOT Mover;
END_TRANSITION
STEP F1Done:
    Done(N);
END_STEP
TRANSITION FROM F1Done TO A6Init
    := Ack;
END_TRANSITION

END_FUNCTION_BLOCK

// ---- L2 Module Controllers/L2_PlatoDivisor_SFC.TcPOU
FUNCTION_BLOCK L2_PlatoDivisor_SFC EXTENDS L1_ControllerBase_SFC

VAR_INPUT 					// Sensores y comandos
	d0  		: BOOL; 
END_VAR

VAR_OUTPUT					// Actuadores
	D_1 		: BOOL; 
    E_1 		: BOOL; 
END_VAR

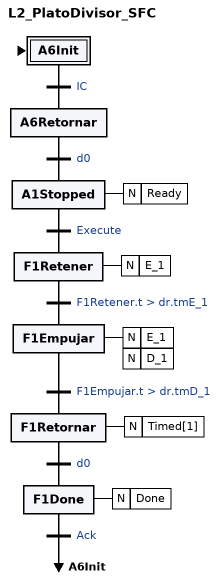
INITIAL_STEP A6Init:
END_STEP
TRANSITION FROM A6Init TO A6Retornar
    := IC;
END_TRANSITION
STEP A6Retornar:
END_STEP
TRANSITION FROM A6Retornar TO A1Stopped
    := d0;
END_TRANSITION
STEP A1Stopped:
    Ready(N);
END_STEP
TRANSITION FROM A1Stopped TO F1Retener
    := Execute;
END_TRANSITION
STEP F1Retener:
    E_1(N);
END_STEP
TRANSITION FROM F1Retener TO F1Empujar
    := F1Retener.t > dr.tmE_1;
END_TRANSITION
STEP F1Empujar:
    E_1(N);
    D_1(N);
END_STEP
TRANSITION FROM F1Empujar TO F1Retornar
    := F1Empujar.t > dr.tmD_1;
END_TRANSITION
STEP F1Retornar:
    Timed[1](N);
END_STEP
TRANSITION FROM F1Retornar TO F1Done
    := d0;
END_TRANSITION
STEP F1Done:
    Done(N);
END_STEP
TRANSITION FROM F1Done TO A6Init
    := Ack;
END_TRANSITION

END_FUNCTION_BLOCK

// ---- L2 Module Controllers/L2_Simple_SFC.TcPOU
FUNCTION_BLOCK L2_Simple_SFC EXTENDS L1_ControllerBase_SFC
// Grafcet simple para los detectores fotoeléctrico e inductivo

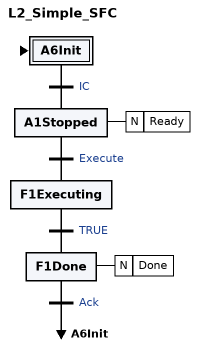
INITIAL_STEP A6Init:
END_STEP
TRANSITION FROM A6Init TO A1Stopped
    := IC;
END_TRANSITION
STEP A1Stopped:
    Ready(N);
END_STEP
TRANSITION FROM A1Stopped TO F1Executing
    := Execute;
END_TRANSITION
STEP F1Executing:
END_STEP
TRANSITION FROM F1Executing TO F1Done
    := TRUE;
END_TRANSITION
STEP F1Done:
    Done(N);
END_STEP
TRANSITION FROM F1Done TO A6Init
    := Ack;
END_TRANSITION

END_FUNCTION_BLOCK

// ---- L3 Modules/L3_Alimentador.TcPOU
FUNCTION_BLOCK L3_Alimentador EXTENDS L1_ModuleBase
(*  MÓDULO ALIMENTACIÓN - Manual de usuario #31/27

Para el almacenamiento y posterior alimentación de las tapas, se utiliza un 
cargador de gravedad, provisto de un empujador accionado mediante cilindro 
neumático que realiza la extracción  *)
VAR_INPUT
	Alimentar		: BOOL;
END_VAR

VAR_OUTPUT	
	fbController	: L2_Alimentador_SFC:=(dr:=dr);	
	k1 				: L1_Sensor;
	K_1 			: L1_Actuator;
	FM 				: L1_Actuator; 
	//_TapaAlimentada	: BOOL;
	FaltaMaterial	: BOOL;
	// Position		: REAL:= 0;
	Leyendo			: BOOL;
END_VAR

METHOD ProcessCycle : BOOL 
VAR_INPUT	
	dr			: REFERENCE TO L1_Director;
	tapas		: REFERENCE TO L6_Tapas;
		
END_VAR
IF dr.gmModeActual = L1_GEMMA.A6Inicializando THEN
	//_TapaAlimentada 			:= FALSE;
	FaltaMaterial				:= FALSE;
ELSE
	// Sensores y condiciones iniciales
	k1.ProcessCycle(LocalHost:=dr.gmLocalHost, sfcValue=>fbController.k1);
	IC:=TRUE; 

	// Controlador
	fbController.ProcessCycle(dr.gmModeActual);
	fbController(Alimentar:=Alimentar, dr:=dr, IC:=IC, Leyendo=>Leyendo, Execute:=Execute, Ack:=Ack, Ready=>Ready, Done=>Done);
	
	// Actuadores y actualización de tapas
	IF Ready AND NOT tapas.EstaAlimentada THEN // 	TapaAlimentada THEN 
		tapas.MoverAlime(Delta:=0); // 	Position := 0;												// Inicialmente la posición es arriba
	ELSIF fbController.Leyendo AND NOT fbController.Performed THEN
		fbController.Performed	:= TRUE;
		FaltaMaterial			:= k1.uiValue;
		//_TapaAlimentada 		:= NOT FaltaMaterial;
		tapas.EstaAlimentada	:= NOT FaltaMaterial;
	ELSIF Done AND NOT fbController.Performed AND Alimentar THEN
		tapas.MoverAlime(Delta:=MoverMax);// Position				:= MaxPosAlime;						// Posición final junto al brazo de carga 
	ELSIF fbController.Executing AND Alimentar THEN // Position < MaxPosAlime AND 
		tapas.MoverAlime(Delta:=1); // Position := Position + 1;									// animación de tapa moviendo hacia abajo		
	END_IF	
	K_1.ProcessCycle(gmMode:=dr.gmModeActual, sfcValue:=fbController.K_1);
	FM.ProcessCycle (gmMode:=dr.gmModeActual, sfcValue:=FaltaMaterial AND dr.Tic);
END_IF
END_METHOD

END_FUNCTION_BLOCK

// ---- L6 Station/L6_Tapas.TcPOU
FUNCTION_BLOCK L6_Tapas
VAR CONSTANT
	ColSecIndeterm	: DWORD := 16#80101010; // gris claro
	ColSecVacio		: DWORD := 16#80808080; // gris oscuro
	ColSecPendiente : DWORD := 16#80000080; // azul
	ColSecDescargar	: DWORD := 16#80008000; // verde
	ColSecEvacuar	: DWORD := 16#80800000; // rojo
END_VAR

VAR_INPUT
	ReqNumero	: DINT := 5; 		// requisito de número de tapas deseadas
	ReqAlta		: REAL := 18.5;  	// requisito de tapa alta
	ReqVacio	: REAL := 2.0; 		// si mide menos el sector está vacío

	ReqAluBaja	: BOOL := TRUE;
	ReqAluAlta	: BOOL := TRUE;
	ReqBlnBaja  : BOOL := TRUE;
    ReqBlnAlta  : BOOL := TRUE;
	ReqNgrBaja  : BOOL := FALSE;
    ReqNgrAlta  : BOOL := FALSE; 

	ResPend	  	: DINT := 0;
	ResReal		: DINT := 0;
	ResRech   	: DINT := 0;
END_VAR

(*
VAR_OUTPUT
	FaltaMat	: BOOL; 
	ExeAlime	: BOOL;	
	AckAlime	: BOOL;
	ExeCarga	: BOOL;
	AckCarga	: BOOL;
	ExeMedid	: BOOL;
	ExeFotoe	: BOOL;
	ExeInduc	: BOOL;
	ExeEvacu	: BOOL;
	AckEvacu	: BOOL;
	ExeDesca	: BOOL;
	AckDesca	: BOOL;
	ExeDescaAnt	: BOOL;
	ExePlato	: BOOL;
	AckPlato	: BOOL;
	ExeSitua	: BOOL;
	ExeTrans	: BOOL;
END_VAR
*)


VAR
	_AlimeEsta	: BOOL; // Esta alimentada o no
	_CargaEsta	: BOOL;
	_DescaEsta	: BOOL;
	
	AlimeY		: REAL; // posición vertical de la tapa alimentándose
	CargaX		: REAL; 
	DescaX		: REAL:=MaxCintaX;
	DescaY		: REAL:=MaxDescaY;
	CintaX		: REAL:=MaxCintaX;
	
	
	//NumGiros 	: DINT := 0;
	PosCarga	: DINT;
	PosFotoe	: DINT;
	PosMedid	: DINT;
	PosInduc	: DINT;
	PosEvacu	: DINT;
	PosDesca	: DINT;
	Alimentada	: BOOL; // HAY UNA TAPA EN EL ALIMENTADOR ESPERANDO A SER CARGADA

	//angulo	 	: REAL := 0.0;
	//anguloanim 	: REAL := 0.0; // angulo para animación que gira lentamente
	//HaGirado	: BOOL := FALSE;
	//Falta_Material		: BOOL;

	vEvacuar_Tapa		: ARRAY[0..7] OF BOOL;
	vDescargar_Tapa		: ARRAY[0..7] OF BOOL;
	
	vInicializando 		: ARRAY[0..7] OF BOOL;	
	//vCargar_Tapa		: ARRAY[0..7] OF BOOL;
	vTapa_Cargada 		: ARRAY[0..7] OF BOOL;
	vAltura_Medida		: ARRAY[0..7] OF BOOL;
	vAltura_Pulsos 		: ARRAY[0..7] OF DWORD;
	vAltura_Mm 			: ARRAY[0..7] OF REAL;
	vTapa_Alta			: ARRAY[0..7] OF BOOL;
	vClaridad_Medida	: ARRAY[0..7] OF BOOL;
	vTapa_Clara 		: ARRAY[0..7] OF BOOL;	
	vMateral_Medido		: ARRAY[0..7] OF BOOL;	
	vTapa_Metalica 		: ARRAY[0..7] OF BOOL;	
	vstrUi 				: ARRAY[0..7] OF STRING;
	vstrToolTip			: ARRAY[0..7] OF STRING;
	vColorSector		: ARRAY[0..7] OF DWORD;
	
	vColorFill			: ARRAY[0..7] OF DWORD;
	vColorFont			: ARRAY[0..7] OF DWORD;	
	vColorFrame			: ARRAY[0..7] OF DWORD;

	Evacu_strUi			: STRING;
	Evacu_strToolTip	: STRING;	
	Evacu_ColorFont		: DWORD;
	Evacu_ColorFrame	: DWORD;
	Evacu_ColorFill		: DWORD;
	Evacu_PosX			: REAL;
	Evacu_PosY			: REAL;
	
	Desca_strUi			: STRING;
	Desca_strToolTip	: STRING;	
	Desca_ColorFont		: DWORD;
	Desca_ColorFrame	: DWORD;
	Desca_ColorFill		: DWORD;
	Desca_PosX			: REAL;
	Desca_PosY			: REAL;

	
END_VAR

METHOD Actualizar : BOOL
VAR_INPUT
END_VAR

VAR
	i 	: INT := 0;
END_VAR

FOR i:=0 TO 7 DO
	vstrTooltip[i] := CONCAT('Sector ', TO_STRING(i));
	vstrTooltip[i] := CONCAT(vstrTooltip[i], ' :');
	IF vInicializando[i] THEN
		vAltura_Medida[i]	:= FALSE;
		vAltura_Pulsos[i]	:= 0;
		vAltura_Mm[i] 		:= 0;
	
		vClaridad_Medida[i]	:= FALSE;
		vTapa_Clara[i] 		:= FALSE;
	
		vMateral_Medido[i]	:= FALSE;	
		vTapa_Metalica[i] 	:= FALSE;
	
		//vCargar_Tapa[i]		:= FALSE;
		vEvacuar_Tapa[i]	:= FALSE;
		vDescargar_Tapa[i]	:= FALSE;	
		vColorSector[i] 	:= ColSecIndeterm;
		vstrUi[i] 			:= '?';
		vstrTooltip[i] 		:= CONCAT(vstrTooltip[i], ' Contenido desconocido => Medir');
		
	ELSIF NOT vTapa_Cargada[i] THEN
		//vCargar_Tapa[i]		:= TRUE;
		vEvacuar_Tapa[i]	:= FALSE;
		vDescargar_Tapa[i]	:= FALSE;	
		vColorSector[i] 	:= ColSecVacio;
		vstrUi[i] 			:= '___';
		vstrTooltip[i] 	:= CONCAT(vstrTooltip[i], ' Sector vacío => Cargar');

	ELSE
		IF vAltura_Medida[i] THEN //  AND vTapa_Cargada[i] redundante porque se cumple
			vstrTooltip[i] 	:= CONCAT(vstrTooltip[i], SEL(vTapa_Alta[i], ' Baja (', ' Alta ('));
			vstrTooltip[i] 	:= CONCAT(vstrTooltip[i], TO_STRING(vAltura_Pulsos[i]));
			vstrTooltip[i] 	:= CONCAT(vstrTooltip[i], ' pulsos, ');
			vstrTooltip[i]	:= CONCAT(vstrTooltip[i], TO_STRING(vAltura_Mm[i]));
			vstrTooltip[i] 	:= CONCAT(vstrTooltip[i], ' mm);');
		ELSE
			vstrTooltip[i] 	:= CONCAT(vstrTooltip[i], ' ¿altura?;');
		END_IF
		
		IF vClaridad_Medida[i] THEN
			vstrTooltip[i] 	:= CONCAT(vstrTooltip[i], SEL(vTapa_Clara[i], ' oscura;', ' clara;'));
		ELSE
			vstrTooltip[i] 	:= CONCAT(vstrTooltip[i], ' ¿claridad?;');							
		END_IF
		IF vMateral_Medido[i] THEN
			vstrTooltip[i] 	:= CONCAT(vstrTooltip[i], SEL(vTapa_Metalica[i], ' plástico;', ' metal;'));
		ELSE
			vstrTooltip[i] 	:= CONCAT(vstrTooltip[i], ' ¿material?;');							
		END_IF
		
		IF vAltura_Medida[i] AND vClaridad_Medida[i] AND vMateral_Medido[i] THEN
			vDescargar_Tapa[i] := (
					(ReqAluAlta AND vTapa_Metalica[i] AND vTapa_Alta[i]) OR
					(ReqAluBaja AND vTapa_Metalica[i] AND NOT vTapa_Alta[i]) OR
					(ReqBlnAlta AND NOT vTapa_Metalica[i] AND vTapa_Clara[i]  AND vTapa_Alta[i]) OR
					(ReqBlnBaja AND NOT vTapa_Metalica[i] AND vTapa_Clara[i]  AND NOT vTapa_Alta[i]) OR
					(ReqNgrAlta AND NOT vTapa_Metalica[i] AND NOT vTapa_Clara[i]  AND vTapa_Alta[i]) OR
					(ReqNgrBaja AND NOT vTapa_Metalica[i] AND NOT vTapa_Clara[i]  AND NOT vTapa_Alta[i]));
			vEvacuar_Tapa[i] := NOT vDescargar_Tapa[i];
			vColorSector[i] := SEL(vDescargar_Tapa[i],ColSecEvacuar, ColSecDescargar);
			vstrTooltip[i] := CONCAT(vstrTooltip[i], SEL(vDescargar_Tapa[i], ' => Evacuar', '=> Descargar'));
		ELSE
			vDescargar_Tapa[i]	:= FALSE;
			vEvacuar_Tapa[i]	:= FALSE;
			vColorSector[i] 	:= ColSecPendiente; 			
			vstrTooltip[i] 		:= CONCAT(vstrTooltip[i], '=> Esperar');
		END_IF 
		vstrUi[i] := SEL(vAltura_Medida[i],'?', SEL(vTapa_Alta[i], 'B','A'));
		vstrUi[i] := CONCAT(vstrUi[i], SEL(vClaridad_Medida[i], '?',SEL(vTapa_Clara[i],'O','C')));
		vstrUi[i] := CONCAT(vstrUi[i], SEL(vMateral_Medido[i], '?', SEL(vTapa_Metalica[i], 'P','M'))); 		
	END_IF
	
	IF vInicializando[i] THEN								// caso A ?
		vColorFill[i]		:= colDesFill;
		vColorFont[i]		:= colDesFont;
		vColorFrame[i]		:= colDesFrameSin;
	ELSIF NOT vTapa_Cargada[i] THEN							// Caso B ___
		vColorFill[i]		:= colVacFill;
		vColorFont[i]		:= colVacFont;
		vColorFrame[i]		:= colVacFrameSin;
	ELSIF NOT vClaridad_Medida[i] THEN						// Caso C A??
		vColorFill[i]		:= colTapFill;
		vColorFont[i]		:= colTapFont;
		vColorFrame[i]		:= colTapFrameSin;
	ELSIF vTapa_Clara[i] AND NOT vMateral_Medido[i] THEN	// Caso D AC?
		vColorFill[i]		:= colClaFill;
		vColorFont[i]		:= colClaFont;
		vColorFrame[i]		:= colClaFrameSin;
	ELSIF NOT vTapa_Clara[i] AND NOT vMateral_Medido[i] THEN // Caso E AO?
		vColorFill[i]		:= colClaFill;
		vColorFont[i]		:= colClaFont;
		vColorFrame[i]		:= colClaFrameSin;
	ELSIF vTapa_Clara[i] AND vTapa_Metalica[i] THEN 		// Caso F ACM
		vColorFill[i]		:= colAluFill;
		vColorFont[i]		:= colAluFont;
		vColorFrame[i]		:= colAluFrameSin;
	ELSIF vTapa_Clara[i] AND NOT vTapa_Metalica[i] THEN 	// Caso G ACP
		vColorFill[i]		:= colBlnFill;
		vColorFont[i]		:= colBlnFont;
		vColorFrame[i]		:= colBlnFrameSin;
	ELSIF NOT vTapa_Clara[i] AND NOT vTapa_Metalica[i] THEN // Caso G AOP
		vColorFill[i]		:= colNgrFill;
		vColorFont[i]		:= colNgrFont;
		vColorFrame[i]		:= colNgrFrameSin;
	ELSE
		vColorFill[i]		:= colErrFill;
		vColorFont[i]		:= colErrFont;
		vColorFrame[i]		:= colErrFrameSin;		
	END_IF
	IF vDescargar_Tapa[i] THEN
		vColorFrame[i]		:= colAluFrameOk; // se aplica el mismo independientemente del tipo de tapa!	
	END_IF
	IF vEvacuar_Tapa[i] THEN
		vColorFrame[i]		:= colAluFrameKo; // se aplica el mismo independientemente del tipo de tapa!			
	END_IF
END_FOR 
ResPend := ReqNumero - ResReal;
END_METHOD

METHOD DebeMedir : BOOL
VAR_INPUT
END_VAR
DebeMedir := not vAltura_Medida[PosMedid];
END_METHOD

PROPERTY EstaAlimentada : BOOL
GET
EstaAlimentada := _AlimeEsta;
END_GET
SET
_AlimeEsta := EstaAlimentada;
END_SET
END_PROPERTY

PROPERTY EstaCargada : BOOL
GET
EstaCargada := _CargaEsta;
END_GET
SET
_CargaEsta := EstaCargada;
END_SET
END_PROPERTY

PROPERTY EstaDescargada : BOOL
GET
EstaDescargada := _DescaEsta;
END_GET
SET
_DescaEsta := EstaDescargada;
END_SET
END_PROPERTY

METHOD Inicializar : BOOL

VAR
	i : DINT;
END_VAR
_AlimeEsta		:= FALSE;
_DescaEsta		:= FALSE;
_CargaEsta		:= FALSE;
AlimeY			:= 0;
CargaX			:= 0;
DescaX			:= MaxCintaX; // oculta como después de transferir
DescaY			:= MaxDescaY;
CintaX			:= MaxCintaX;


ReqAluBaja		:= TRUE;
ReqAluAlta		:= TRUE;
ReqBlnBaja  	:= TRUE;
ReqBlnAlta  	:= TRUE;
ReqNgrBaja  	:= TRUE;
ReqNgrAlta  	:= TRUE; 
Alimentada 		:= FALSE;

ResPend	  		:= 0;
ResReal			:= 0;
ResRech   		:= 0;

//NumGiros	 	:= 0;
//FaltaMat		:= FALSE;
PosMedid 		:= 6; // (NumGiros+6) MOD 8;
PosFotoe 		:= 5; // (NumGiros+5) MOD 8;
PosInduc 		:= 4; // (NumGiros+4) MOD 8;
PosEvacu 		:= 2; // (NumGiros+2) MOD 8;
PosDesca		:= 1; // (NumGiros+1) MOD 8;
PosCarga		:= 0; //(NumGiros+0) MOD 8;

//angulo	 		:= 0.0;
//anguloanim 		:= 0.0; // angulo para animación que gira lentamente
//HaGirado		:= FALSE;
//ExePlato		:= FALSE;


FOR i:=0 TO 7 DO
		vInicializando[i] 	:= TRUE;
END_FOR
Actualizar();
END_METHOD

METHOD MoverAlime : BOOL
VAR_INPUT
	Delta		: REAL;
END_VAR
AlimeY := SEL(Delta=0, SEL(AlimeY > MaxAlimeY or Delta=MoverMax, AlimeY+Delta, MaxAlimeY), 0);
END_METHOD

METHOD MoverCinta : BOOL
VAR_INPUT
	Delta		: REAL;
	Situar		: BOOL;
END_VAR
IF Situar THEN
	CintaX := SEL(Delta=0, SEL(CintaX >= 0 OR Delta=MoverMax, CintaX+Delta, 0), -MinCintaX);
ELSE // transferir
	CintaX := SEL(Delta=0, SEL(CintaX >= MaxCintaX OR Delta=MoverMax, CintaX+Delta, MaxCintaX), 0);
	DescaX := CintaX;
END_IF
END_METHOD

METHOD MoverPickAndPlace : BOOL
VAR_INPUT
	Name		: STRING;
	Delta		: REAL;
END_VAR
IF Name='Carga' THEN
	CargaX := SEL(Delta=0, SEL(CargaX > MaxCargaX OR Delta=MoverMax, CargaX+Delta, MaxCargaX), 0);
ELSE
	DescaX := 0;
	DescaY := SEL(Delta=0, SEL(DescaY > MaxDescaY OR Delta=MoverMax, DescaY+Delta, MaxDescaY), 0);	
END_IF
END_METHOD

METHOD PostDesca : BOOL
ResReal 			:= ResReal + 1;
ResPend				:= ReqNumero - ResReal;

Desca_strUi			:= vstrUi[PosDesca];
Desca_strToolTip	:= vstrToolTip[PosDesca];
Desca_ColorFont		:= vColorFont[PosDesca];
Desca_ColorFrame	:= vColorFrame[PosDesca];
Desca_ColorFill		:= vColorFill[PosDesca];
Desca_PosX			:= 0;
Desca_PosY			:= 0;
Vaciar(PosVacia	:= PosDesca);	
(*
	Desca_strUi			: STRING;
	Desca_strToolTip	: STRING;	
	Desca_ColorFont		: DWORD;
	Desca_ColorFrame	: DWORD;
	Desca_ColorFill		: DWORD;
	Desca_PosX			: REAL;
	Desca_PosY			: REAL;

*)
END_METHOD

METHOD PostEvacu : BOOL
ResRech 			:= ResRech + 1;
Evacu_strUi			:= vstrUi[PosEvacu];
Evacu_strToolTip	:= vstrToolTip[PosEvacu];
Evacu_ColorFont		:= vColorFont[PosEvacu];
Evacu_ColorFrame	:= vColorFrame[PosEvacu];
Evacu_ColorFill		:= vColorFill[PosEvacu];
Vaciar(PosVacia	:= PosEvacu);
END_METHOD

METHOD PostFotoe : BOOL
VAR_INPUT
	Tapa_Clara: BOOL;
END_VAR
vClaridad_Medida[PosFotoe]	:= TRUE;
vTapa_Clara[PosFotoe]		:= Tapa_Clara;
END_METHOD

METHOD PostInduc : BOOL
VAR_INPUT
	Tapa_Metalica: BOOL;
END_VAR
vMateral_Medido[PosInduc]	:= TRUE;
vTapa_Metalica[PosInduc]	:= Tapa_Metalica;
END_METHOD

METHOD PostMedid : BOOL
VAR_INPUT
	Altura_Mm			: REAL;
	Altura_Pulsos		: UDINT;	
END_VAR
vInicializando[PosMedid]		:= FALSE;	
IF Altura_Mm < ReqVacio THEN
	Vaciar(PosVacia:=PosMedid);
ELSE
	vTapa_Cargada[PosMedid]		:= TRUE;			
	vAltura_Medida[PosMedid]	:= TRUE;
	vAltura_Pulsos[PosMedid]	:= Altura_Pulsos;
	vAltura_Mm[PosMedid]		:= Altura_mm;
	vTapa_Alta[PosMedid]		:= Altura_mm > ReqAlta;
END_IF
END_METHOD

METHOD PostPickAndPlace : BOOL
VAR_INPUT
	Name		: STRING;
END_VAR
IF Name = 'Carga' THEN
	_AlimeEsta					:= FALSE; 	// ya no hay tapa en el alimentador
	vInicializando[PosCarga]	:= FALSE;		
	vTapa_Cargada[PosCarga]		:= TRUE;
	vAltura_Medida[PosCarga]	:= FALSE;
	vAltura_Pulsos[PosCarga]	:= 0;
	vAltura_Mm[PosCarga] 		:= 0;		
	vClaridad_Medida[PosCarga]	:= FALSE;
	vTapa_Clara[PosCarga] 		:= FALSE;		
	vMateral_Medido[PosCarga]	:= FALSE;	
	vTapa_Metalica[PosCarga] 	:= FALSE;
	
ELSE // Brazo de descarga
	_DescaEsta			:= TRUE;			// ya hay tapa en el carro
	ResReal 			:= ResReal + 1;
	ResPend				:= ReqNumero - ResReal;
	
	Desca_strUi			:= vstrUi[PosDesca];
	Desca_strToolTip	:= vstrToolTip[PosDesca];
	Desca_ColorFont		:= vColorFont[PosDesca];
	Desca_ColorFrame	:= vColorFrame[PosDesca];
	Desca_ColorFill		:= vColorFill[PosDesca];
	Desca_PosX			:= 0;
	Desca_PosY			:= 0;
	Vaciar(PosVacia	:= PosDesca);	
	(*
		Desca_strUi			: STRING;
		Desca_strToolTip	: STRING;	
		Desca_ColorFont		: DWORD;
		Desca_ColorFrame	: DWORD;
		Desca_ColorFill		: DWORD;
		Desca_PosX			: REAL;
		Desca_PosY			: REAL;
	
	*)	
END_IF
END_METHOD

METHOD ProcessCycle : BOOL
VAR_INPUT
	dr				: REFERENCE TO L1_Director;
	pn				: REFERENCE TO L5_Panel;
	NumGiros 		: DINT;
	//TapaDisponible	: BOOL;
	//TapaCargada		: BOOL; // El brazo de carga ha movido la tapa cargada al plato
	//TapaEvacuada	: BOOL;
	//TapaDescargada	: BOOL;
	
	// Falta_Material	: BOOL;
	//Hay_Pale		: BOOL;
	//ctrlF1			: REFERENCE TO L4_FMS205_F1Producir_SFC;
	//ctrlF2			: REFERENCE TO L4_FMS205_F2SeqPrep_SFC;
	//ctrlF3			: REFERENCE TO L4_FMS205_F3SeqFin_SFC;
	//ctrlF6			: REFERENCE TO L4_FMS205_F6Prueba_SFC;
	//Ready			: BOOL;
	//Done			: BOOL;
	
END_VAR


VAR
	F1	: BOOL;
	A2	: BOOL;
	F2	: BOOL;
	F3	: BOOL;
	F4	: BOOL;
	F5	: BOOL;
	F6	: BOOL;
	i	: int;
END_VAR
IF dr.gmModeActual = L1_GEMMA.A6Inicializando THEN
	ReqAluBaja		:= TRUE;
	ReqAluAlta		:= TRUE;
	ReqBlnBaja  	:= TRUE;
	ReqBlnAlta  	:= TRUE;
	ReqNgrBaja  	:= TRUE;
	ReqNgrAlta  	:= TRUE; 

	ResPend	  		:= 0;
	ResReal			:= 0;
	ResRech   		:= 0;

	FOR i:=0 TO 7 DO
		IF dr.cnF3_Finalizar THEN 
			vInicializando[i] 	:= TRUE;
		ELSE
			Vaciar(PosVacia := i);
		END_IF
	END_FOR	
END_IF

PosMedid 			:= (NumGiros+6) MOD 8;					// -------------- Actualizar posiciones
PosFotoe 			:= (NumGiros+5) MOD 8;
PosInduc 			:= (NumGiros+4) MOD 8;
PosEvacu 			:= (NumGiros+2) MOD 8;
PosDesca			:= (NumGiros+1) MOD 8;
PosCarga			:= (NumGiros+0) MOD 8;
Actualizar();		// calcula qué posiciones hay que descargar o evacuar


//F1					:= ctrlf1.Ready AND dr.gmModeActual=L1_GEMMA.F1ProduccionNormal AND NOT dr.EndBatch;
//A2					:= ctrlf1.Ready AND dr.gmModeActual=L1_GEMMA.A2ParaFinCiclo AND NOT dr.EndBatch;
//F2					:= ctrlF2.Ready AND dr.gmModeActual=L1_GEMMA.F2SecuenciaPreparacion;
//F3					:= ctrlF3.Ready AND dr.gmModeActual=L1_GEMMA.F3SecuenciaFinalizacion;
//F6					:= ctrlF6.Ready AND dr.gmModeActual=L1_GEMMA.F6Probando;
//F5					:= pn.swF5_Ejecutar AND dr.gmModeActual=L1_GEMMA.F5VerificacionOrdenada;


//IF TapaEvacuada THEN
	//ResRech 		:= ResRech + 1;
	//Vaciar(PosVacia := PosEvacu);	
//END_IF



//IF F1 OR A2 OR F2 OR F3 OR F6 OR F5 THEN
	//ExeSitua			:= (F1 OR A2 OR F6 OR (F5 AND pn.swF5_Situar)) AND NOT Hay_Pale;
	//ExeAlime			:= (F1 OR A2 OR F6 OR (F5 AND pn.swF5_Alimentar) AND NOT TapaAlimentada);  // Alimentada);
	//ExeCarga			:= (F1 OR A2 OR F6 OR (F5 AND pn.swF5_Cargar)) AND TapaAlimentada AND  //NOT Falta_Material AND Alimentada AND
	//						NOT vInicializando[PosCarga] AND NOT vTapa_Cargada[PosCarga];
	//ExeMedid			:= (F1 OR A2 OR F6 OR (F5 AND pn.swF5_Medir) OR F2);
	//ExeFotoe			:= (F1 OR A2 OR F6 OR (F5 AND pn.swF5_Claridad) OR F2);
	//ExeInduc			:= (F1 OR A2 OR F6 OR (F5 AND pn.swF5_Material) OR F2);
	//ExeEvacu			:= ((F1 OR A2 OR F6 OR (F5 AND pn.swF5_Evacuar)) AND vEvacuar_Tapa[PosEvacu]) OR
		//				   (F3 AND vTapa_Cargada[PosEvacu]);
	//ExeDesca			:= (F1 OR A2 OR F6 OR (F5 AND pn.swF5_Descargar)) AND vDescargar_Tapa[PosDesca];
	//ExePlato			:= (F1 OR A2 OR F6 OR (F5 AND pn.swF5_Girar) OR F2 OR F3);
	//ExeTrans			:= ExeDescaAnt OR (F5 AND pn.swF5_Transferir); // se transfiere si se descargó en la etapa anterior
	
	//IF ctrlf1.Ready AND ctrlF6.Ready THEN // guarda la decisión de descarga para la transferencia del siguiente ciclo
		//ExeDescaAnt		:= ExeDesca; 	
	//END_IF
//ELSE
	//ExeSitua			:= FALSE;
	//ExeAlime			:= FALSE;
	//ExeCarga			:= FALSE;
	//ExeMedid			:= FALSE;
	//ExeFotoe			:= FALSE;
	//ExeInduc			:= FALSE;
	//ExeEvacu			:= FALSE;
	//ExeDesca			:= FALSE;
	//ExePlato			:= FALSE;
	//ExeTrans			:= FALSE;
//END_IF
//*}

//angulo 					:= -45.0 * (NumGiros MOD 8); //  SEL(angulo=0, angulo-45.0, 315.0); // , angulo+45.0, 0);
	
//IF ExePlato AND anguloanim >-35.0 THEN
	//anguloanim 	:= anguloanim - 0.2;	
//END_IF
END_METHOD

METHOD PuedeCargar : BOOL // TRUE SI EL SECTOR DE CARGA ESTÁ VACÍO
PuedeCargar := NOT vInicializando[PosCarga] AND not vTapa_Cargada[PosCarga];
END_METHOD

METHOD PuedeDescargar : BOOL
PuedeDescargar := vDescargar_Tapa[PosDesca];
END_METHOD

METHOD PuedeEvacuar : BOOL // TRUE SI EL SECTOR CONTIENE UNA TAPA INVÁLIDAD EN LA POSICIÓN DE EVACUACIÓN
VAR_INPUT
	gmMode		: L1_GEMMA;
END_VAR
PuedeEvacuar := vEvacuar_Tapa[PosEvacu]  OR (gmMode=L1_GEMMA.F3SecuenciaFinalizacion AND vTapa_Cargada[PosEvacu]);
END_METHOD

METHOD Vaciar : BOOL
VAR_INPUT
	PosVacia: DINT;
END_VAR
vInicializando[PosVacia]	:= FALSE;	
vTapa_Cargada[PosVacia]		:= FALSE;	
vAltura_Medida[PosVacia]	:= FALSE;
vAltura_Pulsos[PosVacia]	:= 0;
vAltura_Mm [PosVacia]		:= 0;	
vClaridad_Medida[PosVacia]	:= FALSE;
vTapa_Clara[PosVacia] 		:= FALSE;
vMateral_Medido[PosVacia]	:= FALSE;	
vTapa_Metalica[PosVacia] 	:= FALSE;
END_METHOD

END_FUNCTION_BLOCK

// ---- L5 Station User Interfaces/L5_Panel.TcPOU
FUNCTION_BLOCK L5_Panel
VAR_INPUT
	dr								: REFERENCE TO L1_Director;

	mdF1Producir					: BOOL := TRUE;
	//mdF6Probar						: BOOL;
	mdF5Funcion						: BOOL;
	mdF4Planta						: BOOL;

	hwAS_AvisadorSonoro		AT %Q*	: BOOL; 
	hwLA_LamparaAlarma		AT %Q*	: BOOL; 
	//hwDPO_DesconectaPO		AT %Q*	: BOOL; 	
	hwLM_LamparaMarcha		AT %Q*	: BOOL;
	hwLS_LamparaStop		AT %Q*	: BOOL;

	swF0_Empezar					: BOOL;
	swF1_Producir					: BOOL := TRUE;
	swF2_Preparar					: BOOL := TRUE;
	swF3_Finalizar					: BOOL := TRUE;
	swF6_Probar						: BOOL;
	
	swF4_Planta						: BOOL; 
	swMensaje						: STRING(255) :='';
END_VAR

VAR
	hwPE_Seta					AT %I*	: BOOL;
	swPE_Seta							: BOOL;
	
	hwPOC_PulsadorReset			AT %I*	: BOOL; // POC Botón azul está pulsado (PO Conectada)
	swPOC_PulsadorReset					: BOOL; 
	
	hwPM_PulsadorMarcha			AT %I*	: BOOL; // PM - Pulsador de marcha (verde)
	swPM_PulsadorMarcha					: BOOL;
	fpPM_PulsadorMarcha					: R_TRIG;
	
	hwPS_PulsadorStop			AT %I*	: BOOL := TRUE; // PS - Pulsador de parada (rojo)
	swPS_PulsadorStop					: BOOL := TRUE; 
	fnPS_PulsadorStop					: F_TRIG; 
	
	hwSM_SelecAutoManual	 	AT %I*	: BOOL; // SM - Selector modo auto/man
	swSM_SelecAutoManual	 			: BOOL; 	

END_VAR


VAR_OUTPUT
	// consignas del panel, resultado de integrar la información que viene del hardware, el estado GEMMA, los temporizadores y flancos, y la interfaz de usuario		
	swF4_Avanza						: BOOL := FALSE;
 	swF4_Retroc						: BOOL := FALSE;	
	
	swF5_Alimentar					: BOOL;
	fpF5_Alimentar					: R_TRIG;  // cuando se pulsa alimentar hay que quitar cargar
	swF5_Situar						: BOOL;
	swF5_Transferir					: BOOL;
	fpF5_Transferir					: R_TRIG; // cuando se pulsa transferir hay que quitar descargar
	swF5_Cargar						: BOOL;
	fpF5_Cargar						: R_TRIG; // cuando se pulsa cargar hay que quitar girar y alimentar
	swF5_Evacuar					: BOOL;
	fpF5_Evacuar					: R_TRIG; // cuando se pulsa evacuar hay que quitar girar
	swF5_Descargar					: BOOL;
	fpF5_Descargar					: R_TRIG; // cuando se pulsa descargar hay que quitar girar y transferir
	swF5_Medir						: BOOL;
	fpF5_Medir						: R_TRIG; // cuano se pulsa medir hay que quitar girar
	swF5_Claridad					: BOOL;
	swF5_Material					: BOOL;
	swF5_Girar						: BOOL;
	fpF5_Girar						: R_TRIG; // cuando se pulsa girar hay que quitar medir, cargar, descargar y evacuar
	swF5_Ejecutar					: BOOL;
	swF5_Ack						: BOOL;
	
END_VAR

VAR
	gmModeName		: STRING 	:= 'Mode A6';
	gmModeDescr		: STRING 	:= 'Inicializando';	
	
//	ttPE_Seta						: STRING := '';

	swA2_FinCiclo					: BOOL;
	swA3_Estado						: BOOL;
	swA6_Inicializar				: BOOL;

	//swF2_Preparar					: BOOL;
	//swF3_Finalizar				: BOOL;	
	//ttF4_Planta						: STRING :='';
	//enF6_Probar						: BOOL;
	//swF6_Probar						: BOOL;
END_VAR

METHOD ProcessCycle : BOOL
VAR_INPUT
	dr				: REFEREnce to L1_Director;
	gmModeActual	: L1_GEMMA;
	tmReinicio 		: TIME; // = dr.tmTiempoReinicio
END_VAR
IF hwPE_Seta OR swPE_Seta THEN
	dr.cnD1_Emergencia 				:= TRUE;
	dr.cnF4_Planta					:= FALSE; // CON LA SETA NO SE PUEDE ENTRAR EN MODO F4
	dr.cnA6_Inicializar 			:= FALSE; 
	swMensaje 						:= 'Parada de emergencia. Desactive la seta y pulse Reset';

ELSIF dr.cnD1_Emergencia AND NOT (hwPE_Seta OR swPE_Seta) THEN	
	IF hwPOC_PulsadorReset OR swPOC_PulsadorReset THEN
		dr.cnD1_Emergencia 			:= FALSE;
		dr.cnA6_Inicializar 		:= TRUE;
		swMensaje 					:= 'Inicializando...';
	ELSE	
		swMensaje 					:= 'Pulse Reset para reinicializar o entre en modo manual';
		dr.cnF4_Planta				:= hwSM_SelecAutoManual OR swSM_SelecAutoManual;		
	END_IF

ELSIF gmModeActual=L1_GEMMA.A1ParadaInicial OR
	  gmModeActual=L1_GEMMA.F2SecuenciaPreparacion OR
	  gmModeActual=L1_GEMMA.F1ProduccionNormal OR 
	  gmModeActual=L1_GEMMA.F3SecuenciaFinalizacion OR
	  gmModeActual=L1_GEMMA.A2ParaFinCiclo OR	  
	  gmModeActual=L1_GEMMA.F6Probando THEN
	  
	fpPM_PulsadorMarcha(CLK:=hwPM_PulsadorMarcha OR  swPM_PulsadorMarcha);
	fnPS_PulsadorStop  (CLK:=hwPS_PulsadorStop   AND swPS_PulsadorStop);
	IF fpPM_PulsadorMarcha.Q THEN
		dr.cnF0_Empezar 			:= TRUE;
		dr.cnF1_Producir			:= swF1_Producir AND NOT swF6_Probar;
		dr.cnF2_Preparar 			:= swF2_Preparar AND NOT swF6_Probar;
		dr.cnF3_Finalizar			:= swF3_Finalizar AND NOT swF6_Probar;
		dr.cnF6_Probar				:= swF6_Probar AND NOT (swF1_Producir OR swF2_Preparar OR swF3_Finalizar);
	
	ELSIF (hwSM_SelecAutoManual OR swSM_SelecAutoManual) AND NOT DR.cnF4_Planta THEN // paso al modo F4
		dr.cnF4_Planta				:= TRUE;
		dr.cnF1_Producir			:= FALSE;
		dr.cnF6_Probar				:= FALSE;
		dr.cnF5_Funcion				:= FALSE;
		mdF1Producir				:= FALSE;
		mdF5Funcion					:= FALSE;
		swMensaje					:= 'Modo mando directo activado';

	ELSIF mdF1Producir AND NOT dr.cnF1_Producir THEN								// vuelta del modo F4
		dr.cnF4_Planta				:= FALSE;
		swF4_Planta					:= FALSE;
		//dr.cnA2_FinCiclo			:= fnPS_PulsadorStop.Q AND dr.cnF1_Producir AND NOT dr.cnF2_Preparar AND NOT dr.cnF3_Finalizar;
				
		dr.cnF1_Producir			:= swF1_Producir AND NOT swF6_Probar;
		dr.cnF2_Preparar 			:= swF2_Preparar AND NOT swF6_Probar;
		dr.cnF3_Finalizar			:= swF3_Finalizar AND NOT swF6_Probar;
		dr.cnF6_Probar				:= swF6_Probar AND NOT (swF1_Producir OR swF2_Preparar OR swF3_Finalizar);		
		swMensaje					:= 'Modo producción activado';
		
	
		
	ELSIF mdF5Funcion AND NOT dr.cnF5_Funcion THEN
		dr.cnF4_Planta				:= FALSE;
		swF4_Planta					:= FALSE;
		dr.cnF5_Funcion				:= TRUE;
		swMensaje					:= 'Modo función activado';
	END_IF

ELSIF gmModeActual=L1_GEMMA.F4VerificacionSinOrden THEN
	IF NOT (hwSM_SelecAutoManual OR swSM_SelecAutoManual) THEN
		dr.cnF4_Planta				:= FALSE;
		swMensaje					:= 'Modo F4 desactivado';
	END_IF

ELSIF gmModeActual=L1_GEMMA.F5VerificacionOrdenada THEN
	IF NOT mdF5Funcion OR NOT mdF5Funcion OR hwSM_SelecAutoManual OR swSM_SelecAutoManual THEN
		dr.cnF5_Funcion				:= FALSE;
		mdF5Funcion					:= FALSE;
		IF hwSM_SelecAutoManual OR swSM_SelecAutoManual THEN
			dr.cnF4_Planta			:= TRUE;
			swMensaje					:= 'Modo F4 activado';
		ELSE
			swMensaje					:= 'Modo F5 desactivado';			
		END_IF
		
	ELSE
 		fpF5_Alimentar				(CLK := swF5_Alimentar);
		fpF5_Cargar					(CLK := swF5_Cargar);
		fpF5_Medir					(CLK := swF5_Medir);
		fpF5_Evacuar				(CLK := swF5_Evacuar);
		fpF5_Descargar				(CLK := swF5_Descargar);
		fpF5_Girar					(CLK :=swF5_Girar);
		fpF5_Transferir				(CLK :=swF5_Transferir);
		IF fpF5_Alimentar.Q AND swF5_Cargar THEN
			swF5_Cargar				:= FALSE; 
			swMensaje				:= 'No se puede cargar si se alimenta';
		ELSIF fpF5_Cargar.Q AND (swF5_Alimentar OR swF5_Girar)THEN
			swF5_Alimentar			:= FALSE; 
			swF5_Girar				:= FALSE;
			swMensaje				:= 'No se puede alimentar ni girar si se carga';		
		ELSIF fpF5_Medir.Q AND swF5_Girar THEN
			swF5_Girar				:= FALSE; 
			swMensaje				:= 'No se puede girar si se mide';
		ELSIF fpF5_Evacuar.Q AND swF5_Girar THEN	
			swF5_Girar				:= FALSE; 
			swMensaje				:= 'No se puede girar si se evacúa';
		ELSIF fpF5_Descargar.Q AND (swF5_Girar OR swF5_Transferir) THEN
			swF5_Girar				:= FALSE; 
			swF5_Transferir			:= FALSE;
			swMensaje				:= 'No se puede girar ni transferir si se descarga';
		ELSIF fpF5_Girar.Q AND (swF5_Cargar OR swF5_Medir OR swF5_Evacuar OR swF5_Descargar) THEN
			swF5_Cargar				:= FALSE;
			swF5_Medir				:= FALSE;
			swF5_Evacuar			:= FALSE;
			swF5_Descargar			:= FALSE;
			swMensaje				:= 'No se puede cargar, medir, evacuar ni descargar si se gira';
		ELSIF fpF5_Transferir.Q AND swF5_Descargar THEN
			swF5_Descargar			:= FALSE; 
			swMensaje				:= 'No se puede descargar si se transfiere';
		END_IF		
	END_IF

	 
ELSE
	(*

ttPE_Seta := 'Pulsar la seta o el botón para parada de emergencia';	
ttF4_Planta := 'Mandos directos desactivados';
FP_PM(CLk := hwPM_PulsadorMarcha);

dr.cnA1_ParadaIni := FALSE;
	dr.cnA6_Inicializar := FALSE; 
	dr.cnF4_Planta 		:= FALSE;
	dr.cnF5_Funcion 	:= FALSE;
	dr.cnF6_Probar 		:= FALSE;
	dr.cnF1_Producir	:= FALSE;

//----------------------------------------------------------------- Consiga cnD1_Emergencia
dr.cnD1_Emergencia := hwPE_Seta OR swPE_Seta; 
IF dr.cnD1_Emergencia THEN
	IF hwPE_Seta THEN
		IF swPE_Seta THEN
			ttPE_Seta := 'Desarmar la seta y desactivar el botón para reinicializar';
		ELSE
			ttPE_Seta := 'Desarmar la seta para reinicializar';		
		END_IF
	ELSE
		IF swPE_Seta THEN
			ttPE_Seta := 'Desactivar el botón para reinicializar';
		END_IF
	END_IF

//----------------------------------------------------------------- Consigna A6_Inicializar
ELSIF swA6_Inicializar THEN //  OR TmpReinicio.Q);
	// TmpReinicio(IN := hwPM_PulsadorMarcha AND NOT hwPS_PulsadorStop, PT:= tmReinicio);
	dr.cnA6_Inicializar := TRUE; 
	//mdF1Producir := FALSE;
	//mdF4Planta := FALSE;
	//mdF5Funcion := FALSE;
	//mdF6Probar := FALSE;
 
	
//----------------------------------------------------------------- Modo F4_Planta
ELSIF (hwSM_SelecAutoManual OR mdF4Planta) THEN 
	//mdF1Producir 	:= FALSE;
	dr.cnF4_Planta 	:= TRUE;
	//dr.cnF5_Funcion := TRUE;
	//mdF5Funcion 	:= FALSE;
	//mdF6Probar 		:= FALSE;
	IF hwSM_SelecAutoManual AND swF4_Planta THEN
		ttF4_Planta := 'Mandos directos ativados desde panel físico y visualización';
	ELSIF hwSM_SelecAutoManual THEN	
		ttF4_Planta := 'Mandos directos ativados desde panel físico';
	ELSIF swF4_Planta THEN
		ttF4_Planta := 'Mandos directos ativados desde visualización';
	END_IF	

	
	

//----------------------------------------------------------------- F5_Funcion
ELSIF mdF5Funcion THEN  
	//mdF1Producir 	:= FALSE;
	//mdF4Planta 		:= FALSE;
	dr.cnF5_Funcion := TRUE;
	//mdF6Probar 		:= FALSE;

	IF swF5_Girar AND (swF5_Cargar OR swF5_Evacuar OR swF5_Descargar OR swF5_Medir) THEN 
		//swF5_Girar := FALSE;
		swF5_Cargar := FALSE;
		swF5_Evacuar := FALSE;
		swF5_Descargar := FALSE;
		swF5_Medir := FALSE;
		swMensaje := 'No se puede girar a la vez que cargar, evacuar, descargar o medir por riesgo de avería';
	END_IF
	IF swF5_Alimentar AND swF5_Cargar THEN // funciones incompatibles
		swF5_Cargar := FALSE;
		swMensaje := 'No se puede cargar a la vez que alimentar por riesgo de avería';
	END_IF
	IF swF5_Transferir AND swF5_Descargar THEN
		swF5_Transferir := FALSE;
		swMensaje := 'No se puede descargar a la vez que transferer por riesgo de avería';
	END_IF


	
//----------------------------------------------------------------- F6_Probar
ELSIF mdF6Probar THEN  
	//mdF1Producir	:= FALSE;
	//mdF4Planta 		:= FALSE;
	//mdF5Funcion 	:= FALSE;
	dr.cnA1_ParadaIni := NOT dr.cnF0_Empezar;
	dr.cnF6_Probar 	:= TRUE;
	IF (swF0_Empezar OR FP_PM.Q) THEN
		dr.cnF0_Empezar := TRUE;
	END_IF

	
//----------------------------------------------------------------- F1_Producir
ELSIF (mdF1Producir OR FP_PM.Q) THEN
	dr.cnF1_Producir:= TRUE;

	IF (swF0_Empezar OR FP_PM.Q) THEN
		dr.cnF0_Empezar := TRUE;
	END_IF
	//dr.cnF0_Empezar := (swF0_Empezar OR FP_PM.Q);  
	dr.cnA1_ParadaIni := NOT dr.cnF0_Empezar;
	//mdF4Planta 		:= FALSE;
	//mdF5Funcion 	:= FALSE;
	//mdF6Probar	 	:= FALSE;

	dr.cnA2_FinCiclo:= (swA2_FinCiclo OR hwPS_PulsadorStop); // enA2_FinCiclo AND (swA2_FinCiclo OR hwPS_PulsadorStop);
	dr.cnA3_Estado 	:= swA3_Estado;

ELSE
	dr.cnF0_Empezar :=FALSE; 
	//dr.cnA1_ParadaIni 	:= TRUE;
	dr.cnA6_Inicializar := FALSE; 
	dr.cnF4_Planta 		:= FALSE;
	dr.cnF5_Funcion 	:= FALSE;
	dr.cnF6_Probar 		:= FALSE;
	dr.cnF1_Producir	:= FALSE;
END_IF 

IF dr.Failure OR dr.gmModeActual=L1_GEMMA.A4ParadaObtenida OR dr.gmModeActual=L1_GEMMA.D2TratamientoFallos THEN
	dr.cnF0_Empezar := FALSE;
	IF (swF0_Empezar OR FP_PM.Q) THEN
		dr.cnF0_Empezar := TRUE;
	END_IF	
END_IF

(*
dr.cnF1_Empezar := enF1_Empezar AND (swF1_Empezar OR FP_PM.Q);
IF NOT dr.cnF1_Empezar AND (swF1_Empezar OR FP_PM.Q) THEN // consigna no válida
	swF1_Empezar := FALSE; // si no se puede entrar en el modo hay que desactivar el botón
	swMensaje := 'Sólo se puede empezar desde una parada';
END_IF

//----------------------------------------------------------------- Consigna A2_ParaFinCiclo

IF NOT dr.cnA2_FinCiclo AND (swA2_FinCiclo OR hwPS_PulsadorStop) THEN // consigna no válida
	swA2_FinCiclo := FALSE; // si no se puede entrar en el modo hay que desactivar el botón
	swMensaje := 'Sólo se puede pasar a A2 desde el modo F1';

ELS 
IF dr.cnA2_FinCiclo THEN
	// swA2_FinCiclo := TRUE; 
	IF gmModeActual = L1_GEMMA.F1ProduccionNormal THEN
		swMensaje := 'Esperando a finalizar el ciclo para parar';
	ELSIF gmModeActual = L1_GEMMA.A4ParadaObtenida THEN
		swMensaje := 'Parada obtenida después de acabar el ciclo';
	END_IF
END_IF 
dr.cnA3_Estado := enA3_Estado AND (swA3_Estado);
IF NOT dr.cnA3_Estado AND (swA3_Estado) THEN // consigna no válida
	swA3_Estado := FALSE; // si no se puede entrar en el modo hay que desactivar el botón
	swMensaje := 'Sólo se puede pasar a A3 desde el modo F1, F5 o A2';

ELSIF dr.cnA3_Estado THEN
	swA3_Estado := TRUE; 
	IF gmModeActual = L1_GEMMA.A4ParadaObtenida THEN
		swMensaje := 'Parada obtenida después de alcanzar un estado estable';
	ELSE
		swMensaje := 'Esperando a un estado estable para parar';
	END_IF
END_IF

//----------------------------------------------------------------- Consigna F1_Reanudar
dr.cnF1_Reanudar := enF1_Reanduar AND (swF1_Reanudar OR hwPM_PulsadorMarcha);
 	
IF NOT dr.cnF1_Reanudar AND (swF1_Reanudar OR hwPM_PulsadorMarcha) THEN // consigna no válida
	swF1_Reanudar := FALSE; // si no se puede entrar en el modo hay que desactivar el botón
	swMensaje := 'Sólo se puede reanudar desde una parada';

ELSIF dr.cnF1_Reanudar THEN
	swMensaje := 'Reanundando tras la parada';
END_IF

//----------------------------------------------------------------- Consigna A3_Estado
	
*)







*)

//----------------------------------------------------------------- Consigna F1_Empezar

END_IF

UpdateUI(gmMode := dr.gmModeActual);
END_METHOD

METHOD UpdateUi : BOOL
VAR_INPUT
	gmMode				: L1_GEMMA;
END_VAR
// actualizar actuadores del panel
hwAS_AvisadorSonoro 			:= FALSE;
hwLA_LamparaAlarma				:= FALSE;
hwLM_LamparaMarcha				:= FALSE;

CASE gmMode OF
	L1_GEMMA.A1ParadaInicial:
		gmModeName				:= 'Mode A1';
		gmModeDescr				:= 'Parada en estado inicial';
		hwLM_LamparaMarcha		:= dr.Tic;
		
	L1_GEMMA.A2ParaFinCiclo:
		gmModeName				:= 'Mode A2';
		gmModeDescr				:= 'Parada a final de ciclo solicitada';
		hwLM_LamparaMarcha		:= TRUE;
		
	L1_GEMMA.A3ParadaEstado:
		gmModeName				:= 'Mode A3';
		gmModeDescr				:= 'Parada en estado actual solicitada';
		
	L1_GEMMA.A4ParadaObtenida:
		gmModeName				:= 'Mode A4';
		gmModeDescr				:= 'Parada obtenida';
		
	L1_GEMMA.A5PreparandoTrasFallo:
		gmModeName				:= 'Mode A5';
		gmModeDescr				:= 'Preparando tras fallo';	
		
	L1_GEMMA.A6Inicializando:
		gmModeName				:= 'Mode A6';
		gmModeDescr				:= 'Inicializando';
		hwLA_LamparaAlarma		:= dr.Tic;
		//hwDPO_DesconectaPO		:= dr.Tic;
		
	L1_GEMMA.A7SituandoEstado:
		gmModeName				:= 'Mode A7';
		gmModeDescr				:= 'Situando PO en un estado determinado';

	L1_GEMMA.F1ProduccionNormal:
		gmModeName				:= 'Mode F1';
		gmModeDescr				:= 'Producción normal';
		hwLM_LamparaMarcha		:= TRUE;

	L1_GEMMA.F2SecuenciaPreparacion:
		gmModeName				:= 'Mode F2';
		gmModeDescr				:= 'Secuencia de preparación';	
		hwAS_AvisadorSonoro 	:= dr.Tic;
		hwLM_LamparaMarcha		:= TRUE;
		
	L1_GEMMA.F3SecuenciaFinalizacion:
		gmModeName				:= 'Mode F3';
		gmModeDescr				:= 'Secuencia de finalización';
		hwAS_AvisadorSonoro 	:= TRUE;
		hwLM_LamparaMarcha		:= TRUE;
		
	L1_GEMMA.F4VerificacionSinOrden:
		gmModeName				:= 'Mode F4';
		gmModeDescr				:= 'Verificación sin orden (Planta)';
		
	L1_GEMMA.F5VerificacionOrdenada:
		gmModeName				:= 'Mode F5';
		gmModeDescr				:= 'Verificación ordenada (Función)';
				
	L1_GEMMA.F6Probando:
		gmModeName				:= 'Mode F6';
		gmModeDescr				:= 'Probando';
		
	L1_GEMMA.D1ParadaEmergencia:
		gmModeName				:= 'Mode D1';
		gmModeDescr				:= 'Parada de emergencia';
		hwAS_AvisadorSonoro 	:= dr.Tic;
		hwLA_LamparaAlarma		:= dr.Tic;

	L1_GEMMA.D2TratamientoFallos:
		gmModeName				:= 'Mode D2';
		gmModeDescr				:= 'Diagnósdr.tico/tratamiento de fallos';
		hwAS_AvisadorSonoro 	:= dr.Tic;
		hwLA_LamparaAlarma	:= dr.Tic;
		
	L1_GEMMA.D3ProducirConFallos:
		gmModeName				:= 'Mode D3';
		gmModeDescr				:= 'Producir con fallos';

END_CASE
END_METHOD

END_FUNCTION_BLOCK

// ---- L3 Modules/L3_CaptadorInductivo.TcPOU
FUNCTION_BLOCK L3_CaptadorInductivo EXTENDS L1_ModuleBase
(* ESTACIONES DE DETECCIÓN DE MATERIAL - Manual de usuario #31/27

Para poder diferenciar las tapas del primero de estos tipos, la segunda de 
las estaciones del plato divisor está dotada con un captador inductivo. Éste 
proporciona una señal al PLC, únicamente en el caso de que la tapa que el 
plato sitúa frente a él cada vez que realiza un giro, sea de aluminio. *)

VAR_OUTPUT
	fbController		: L2_Simple_SFC:=(dr:=dr);		
	di         			: L1_Sensor;					
	Tapa_Metalica		: BOOL;
	strUi				: STRING := '?';
END_VAR

VAR
	simula		: DRAND := (Seed:=1);
END_VAR

METHOD ProcessCycle : BOOL
VAR_INPUT
	dr			: REFERENCE TO L1_Director;
	tapas		: REFERENCE TO L6_Tapas;	
END_VAR
// Sensores y condiciones iniciales
di.ProcessCycle(LocalHost:=dr.gmLocalHost,);
IC := TRUE;

// Controlador
fbController.ProcessCycle(dr.gmModeActual);
fbController(
	dr:=dr, IC:=IC, Execute:=Execute, Ack:=Ack, Ready=>Ready, Done=>Done);

// Actuadores y actualización de tapas
IF Done AND NOT fbController.Performed THEN //  Lectura_Registrada THEN
	fbController.Performed 	:= TRUE;
	IF dr.gmLocalHost THEN
		simula();
		Tapa_Metalica := SEL (simula.Num < 0.40, FALSE, TRUE); // 40/60% simuladas metálicas/plástico
	ELSE
		Tapa_Metalica		:= di.uiValue;	
	END_IF
	strUi := SEL(Tapa_Metalica, 'Plástico','Metálica');
	tapas.PostInduc(Tapa_Metalica:=Tapa_Metalica);
	
ELSIF Ready THEN // una vez que cambia el ciclo la lectura ya no es fiable	
	strUi := '?';
END_IF
END_METHOD

END_FUNCTION_BLOCK

// ---- L3 Modules/L3_Cinta.TcPOU
FUNCTION_BLOCK L3_Cinta EXTENDS L1_ModuleBase

VAR_INPUT
	Situar			: BOOL;
	Transferir		: BOOL;
END_VAR

VAR_OUTPUT
	fbController			: L2_Cinta_SFC:=(dr:=dr);
	pp						: L1_Sensor;
	cp0						: L1_Sensor;
	cp1						: L1_Sensor;
	cp2						: L1_Sensor;
	RUN						: L1_Actuator;
	REV						: L1_Actuator;
	R_1						: L1_Actuator;
	S_1						: L1_Actuator;
	Carro_Situado			: BOOL;
	Carro_Transfer			: BOOL;
	Position_Carro			: REAL := 0;
	PosDescaX				: REAL := 0;		// posición X de la tapa descargada (0 bajo el plato)
	_TapaDescargada			: BOOL;			
	// tipo de tapa descargada
	

	// colores para distingur cuándo situa y cuándo transfiere	
	colPicFramTransferir 	: DWORD;
	colPicFillTransferir 	: DWORD;

	colPicFramSituar 		: DWORD;
	colPicFillSituar 		: DWORD;
	PosTapaY				: REAL; 
END_VAR


VAR CONSTANT
END_VAR

METHOD ProcessCycle : BOOL 
VAR_INPUT
	dr			: REFERENCE TO L1_Director;
	tapas		: REFERENCE TO L6_Tapas;	
END_VAR
IF dr.gmModeActual = L1_GEMMA.A6Inicializando THEN
	Carro_Situado	 			:= FALSE;
	Carro_Transfer				:= FALSE;
	Position_Carro				:= MinPosCarro; // empieza a la izquierda de la visu
	//PosTapaY					:= 0; // empieza arriba en el plato
ELSE
	// Sensores y condiciones iniciales
	pp.ProcessCycle (LocalHost:=dr.gmLocalHost, sfcValue=>fbController.pp);
	cp0.ProcessCycle(LocalHost:=dr.gmLocalHost, sfcValue=>fbController.cp0);
	cp1.ProcessCycle(LocalHost:=dr.gmLocalHost, sfcValue=>fbController.cp1);
	cp2.ProcessCycle(LocalHost:=dr.gmLocalHost, sfcValue=>fbController.cp2);
	IC := TRUE;
	
	// Controlador
	fbController.ProcessCycle(dr.gmModeActual);
	fbController(Situar := Situar, Transferir := Transferir,	
		dr:=dr, IC:=IC, Execute:=Execute, Ack:=Ack, Ready=>Ready, Done=>Done);
	
	// Actuadores y actualización de tapas
	IF Ready AND NOT Carro_Situado THEN
		tapas.MoverCinta(Delta:=0, Situar:=TRUE);
		//Position_Carro			:= MinPosCarro; // carro a la izquierda
		//PosTapaY				:= 0; // tapa arriba
	ELSIF Ready AND NOT Carro_Transfer THEN
		tapas.MoverCinta(Delta:=0, Situar:=FALSE);
		//Position_Carro			:= 0; // carro bajo el plato
		//PosTapaY				:= SEL(_TapaDescargada, 0, MaxPosTapaY); // tapa arriba o abajo
		//Pos_Situa				:= SEL(Carro_Situado,-MaxPosSitua, 0);
		//Pos_Trans				:= SEL(Carro_Transfer, 0, MaxPosTrans); 
	ELSIF Ready AND Carro_Transfer THEN
		PosDescaX				:=0;	
		Position_Carro			:= MaxPosCarro; // carro a la derecha
		//PosTapaY				:= SEL(_TapaDescargada, 0, MaxPosTapaY); // tapa arriba o abajo
	ELSIF Done AND NOT fbController.Performed AND Situar THEN
		fbController.Performed 	:= TRUE;
		Carro_Situado			:= TRUE;
		Carro_Transfer			:= FALSE;
		_TapaDescargada			:= FALSE;
		tapas.MoverCinta(Delta:=MoverMax, Situar:=TRUE);
		//Position_Carro			:= 0;
		//PosTapaY				:= 0;
	ELSIF Done AND NOT fbController.Performed AND Transferir THEN
		fbController.Performed 	:= TRUE;
		Carro_Transfer			:= TRUE;
		Carro_Situado			:= FALSE;
		//Position_Carro			:= MaxPosCarro; 
		//PosDescaX				:= MaxPosCarro;
		tapas.MoverCinta(Delta:=MoverMax, Situar:=FALSE);	
		_TapaDescargada			:= FALSE;
	//ELSIF fbController.Executing AND Situar AND Position_Carro <0 THEN
		//Position_Carro 			:= Position_Carro + 2;													
	//ELSIF fbController.Executing AND Transferir AND Position_Carro < MaxPosCarro THEN
		//Position_Carro 			:= Position_Carro + 2;
		//PosDescaX				:= SEL(_TapaDescargada, 0, Position_Carro); // al transferir el carro y la tapa se mueven al unísiono
		//		PosTapaY				:= MaxPosTapaY;
	ELSIF fbController.Executing THEN
		tapas.MoverCinta(Delta:=2, Situar:=Situar);									
	END_IF	
	RUN.ProcessCycle(gmMode:=dr.gmModeActual, sfcValue:=fbController.RUN);
	REV.ProcessCycle(gmMode:=dr.gmModeActual, sfcValue:=fbController.REV);
	R_1.ProcessCycle(gmMode:=dr.gmModeActual, sfcValue:=fbController.R_1);
	S_1.ProcessCycle(gmMode:=dr.gmModeActual, sfcValue:=fbController.S_1);

	// Actualizar las flechas de la cinta dependiendo de si sitúa o transfiere
	colPicFramTransferir := SEL(Transferir, colModFramReady, fbController.colPicFram);
	colPicFillTransferir := SEL(Transferir, colModFillReady, fbController.colPicFill);
	colPicFramSituar	 := SEL(Situar, 	colModFramReady, fbController.colPicFram);
	colPicFillSituar	 := SEL(Situar, 	colModFillReady, fbController.colPicFill);
	
END_IF


// tapas.PostCinta(Done := Done, Situa:=Situar, Trans:=Transferir);
END_METHOD

PROPERTY TapaDescargada : bool
GET
TapaDescargada := _TapaDescargada;
END_GET
SET
_TapaDescargada := TapaDescargada;
END_SET
END_PROPERTY

END_FUNCTION_BLOCK

// ---- L3 Modules/L3_DetectorFotoelectrico.TcPOU
FUNCTION_BLOCK L3_DetectorFotoelectrico EXTENDS L1_ModuleBase
(*

ESTACIONES DE DETECCIÓN DE MATERIAL - Manual de usuario #32/28

Con el fin de diferenciar finalmente las tapas de nylon blanco de las de
color negro, se ha incluido un detector fotoeléctrico. Dicho componente 
proporciona una señal de detección únicamente, de las tapas de color 
blanco
 
*)

VAR_OUTPUT
	fbController		: L2_Simple_SFC:=(dr:=dr);
	df 		        	: L1_Sensor;
	Tapa_Clara			: BOOL;
	strUi 				: STRING := '?';
END_VAR

VAR
	simula		: DRAND := (Seed:=1);
END_VAR

METHOD ProcessCycle : BOOL
VAR_INPUT
	dr			: REFERENCE TO L1_Director;
	tapas		: REFERENCE TO L6_Tapas;	
END_VAR
// Sensores y condiciones iniciales
df.ProcessCycle(LocalHost:=dr.gmLocalHost);
IC := TRUE;

// Controlador
fbController.ProcessCycle(dr.gmModeActual);
fbController(
	dr:=dr, IC:=IC, Execute:=Execute, Ack:=Ack, Ready=>Ready, Done=>Done);

// Actuadores y actualización de tapas
IF Done AND NOT fbController.Performed THEN //  Lectura_Registrada THEN // si ha terminado de captar: guardar resultado
	//Lectura_Registrada	:= TRUE;
	fbController.Performed	:= TRUE;
	IF dr.gmLocalHost THEN
		simula();
		Tapa_Clara 			:= SEL (simula.Num < 0.40, TRUE, FALSE); // 40/60% simuladas oscuras/claras
	ELSE
		Tapa_Clara			:= df.uiValue;	
	END_IF

	
	strUi 				:= SEL(Tapa_Clara, 'Oscura','Clara');
	tapas.PostFotoe(Tapa_Clara:=Tapa_Clara);

ELSIF Ready THEN // una vez que cambia el ciclo la lectura ya no es fiable	
	//Lectura_Registrada		:= FALSE;
	strUi := '?';
END_IF
END_METHOD

END_FUNCTION_BLOCK

// ---- L3 Modules/L3_Evacuador.TcPOU
FUNCTION_BLOCK L3_Evacuador EXTENDS L1_ModuleBase
(* 
ESTACIÓN DE EVACUACIÓN DE TAPA INCORRECTA - Manual de usuario #33/29

En caso de que la tapa que llegue a la penúltima de las estaciones del plato divisor, tras haber pasado por 
los diferentes sensores encargados de determinar su material y su altura, no coincida con lo indicado por el 
controlador central encargado de planificar la producción, ha de ser rechazada. Para ello se ha dispuesto en esta 
estación un manipulador de dos ejes que en caso de recibir la orden correspondiente, recoge la tapa del plato 
divisor y la deposita sobre una rampa de evacuación.

Los componentes que forman parte de este manipulador son dos cilindros neumáticos de vástagos paralelos a modo de ejes, 
sobre los que se ha fijado como elemento terminal una placa con tres ventosas para sujeción por vacío

*)

VAR_INPUT
	Evacuar			: BOOL;	
END_VAR

VAR_OUTPUT
	fbController	: L2_Evacuador_SFC:=(dr:=dr);
	f0 				: L1_Sensor;
	f1 				: L1_Sensor := (uiValue:=TRUE);
	g0 				: L1_Sensor;
	v1 				: L1_Sensor;	
	F_0				: L1_Actuator;
	F_1				: L1_Actuator;
	G_1				: L1_Actuator;
	V_1				: L1_Actuator;
	_TapaEvacuada	: BOOL;
	Position		: REAL:= 0;
END_VAR

METHOD ProcessCycle : BOOL 
VAR_INPUT
	dr			: REFERENCE TO L1_Director;
	tapas		: REFERENCE TO L6_Tapas;	
END_VAR
IF dr.gmModeActual = L1_GEMMA.A6Inicializando THEN
	_TapaEvacuada	 			:= FALSE;
ELSE
	// Sensores y condiciones iniciales
	f0.ProcessCycle(LocalHost:=dr.gmLocalHost, sfcValue=>fbController.f0);
	f1.ProcessCycle(LocalHost:=dr.gmLocalHost, sfcValue=>fbController.f1);
	g0.ProcessCycle(LocalHost:=dr.gmLocalHost, sfcValue=>fbController.g0);
	v1.ProcessCycle(LocalHost:=dr.gmLocalHost, sfcValue=>fbController.v1);
	IC := f1.hwValue; // el evacuador está en condiciones iniciales cuando el sensor f1 está activado

	// Controlador
	fbController.ProcessCycle(dr.gmModeActual);
	fbController(Evacuar:=Evacuar, dr:=dr, IC:=IC, Execute:=Execute, Ack:=Ack, Ready=>Ready, Done=>Done);
	IF Ready AND NOT _TapaEvacuada THEN 
		Position := 0;											
	ELSIF Done AND NOT fbController.Performed AND Evacuar THEN
		fbController.Performed 	:= TRUE;
		_TapaEvacuada	 		:= TRUE;
		Position				:= MaxPosEvacu;
		tapas.PostEvacu();						 
	ELSIF fbController.Executing AND Position < MaxPosEvacu AND Evacuar THEN
		Position := Position + 1;											
	END_IF		
	
	// Actuadores y actualización de tapas		
	F_0.ProcessCycle(gmMode:=dr.gmModeActual, sfcValue:=fbController.F_0);
	F_1.ProcessCycle(gmMode:=dr.gmModeActual, sfcValue:=fbController.F_1);
	G_1.ProcessCycle(gmMode:=dr.gmModeActual, sfcValue:=fbController.G_1);
	V_1.ProcessCycle(gmMode:=dr.gmModeActual, sfcValue:=fbController.V_1);


END_IF
END_METHOD

PROPERTY TapaEvacuada : BOOL
GET
TapaEvacuada := _TapaEvacuada;
END_GET
SET
_TapaEvacuada := TapaEvacuada;
END_SET
END_PROPERTY

END_FUNCTION_BLOCK

// ---- L3 Modules/L3_MedidorTapa.TcPOU
FUNCTION_BLOCK L3_MedidorTapa EXTENDS L1_ModuleBase
(*

ESTACIÓN MEDICIÓN TAPA - Manual de usuario #32/28

El hecho de disponer de tapas con dos alturas diferentes hace necesario disponer de un elemento 
que realice una medición de las mismas. Debido a la finalidad didáctica con la cual se ha realizado el
diseño de esta célula, se han adoptado soluciones variadas para llevar a cabo operaciones similares. 
En otras estaciones, para operaciones de medición se ha recurrido a componentes como cilindros 
neumáticos con detectores de altura correcta, o palpadores con salida analógica. En este caso se ha 
considerado de interés utilizar un transductor digital que proporciona una salida por pulsos, como es el 
encoder lineal.

La imagen muestra el aspecto del componente utilizado, el cuál consta 
de un cilindro neumático que desplaza el palpador hasta contactar con la 
tapa, en combinación con un encoder lineal integrado en el mismo cilindro. 
Mediante la cuenta de los pulsos suministrados por el encoder, realizada 
mediante una entrada de contaje rápido del PLC, es posible determinar la 
distancia que avanza al cilindro hasta contactar con la tapa. Disponiendo de 
este dato es posible determinar de forma directa la altura de la tapa

*)

VAR_INPUT
	Medir			: BOOL;	
END_VAR

VAR_OUTPUT
	fbController		: L2_MedidorTapa_SFC:=(dr:=dr);
	dh 			AT %I*	: UINT := 3000; (*Detector valor altura *)
	L_1 				: L1_Actuator;

	//Lectura_Registrada	: BOOL;
	Altura_mm			: REAL;
	Altura_Pulsos		: UINT;
	strUi : STRING 		:= '?';	

END_VAR

VAR
	simula		: DRAND := (Seed:=1);
END_VAR

METHOD ProcessCycle : BOOL 
VAR_INPUT
	dr			: REFERENCE TO L1_Director;
	tapas		: REFERENCE TO L6_Tapas;	
END_VAR
// Sensores y condiciones iniciales
IC := TRUE;

// Controlador
fbController.ProcessCycle(dr.gmModeActual);
fbController(Medir:=Medir, dh := dh, 
	dr:=dr, IC:=IC, Execute:=Execute, Ack:=Ack, Ready=>Ready, Done=>Done);
	
// Actuadores y actualización de tapas
L_1.ProcessCycle(gmMode:=dr.gmModeActual, sfcValue:=fbController.L_1);
IF fbController.Leyendo AND NOT fbController.Performed THEN
	fbController.Performed 	 		:= TRUE;
	IF dr.gmLocalHost THEN // en pruebas sin estación, la altura es un número aleatorio
		simula();
		dh := TO_UINT(simula.Num*2000);
		Altura_mm		:= -0.0257*dh + 52.532;				  // calcular la altura con la ecuación de regresión
		Altura_mm 		:= SEL(Altura_mm < 0, Altura_mm, 10); // simulando siempre hay tapa
	ELSE
		Altura_Pulsos	:= dh;
		Altura_mm		:= -0.0257*dh + 52.532;				 // calcular la altura con la ecuación de regresión
		Altura_mm 		:= SEL(Altura_mm < 0, Altura_mm, 0); // si la altura es negativa dejar cero
	END_IF	

	Altura_mm		:= TO_INT(100*Altura_mm)/100.0; 		// dejar sólo 2 decimales
	strUi := TO_STRING(Altura_mm);
	strUi := concat(strUi, ' mm');
	tapas.PostMedid(Altura_Mm:=Altura_mm, Altura_Pulsos:=Altura_Pulsos);

ELSIF Ready THEN // Resetear la lectura para el siguiente ciclo
	Altura_Pulsos	:= 0;
	Altura_mm		:= 0;
	strUi := '?';
END_IF
END_METHOD

END_FUNCTION_BLOCK

// ---- L3 Modules/L3_PickAndPlace.TcPOU
FUNCTION_BLOCK L3_PickAndPlace EXTENDS L1_ModuleBase
(* ESTACIÓN DE CARGA - Manual de usuario #31/27 
La alimentación de material descrita en el punto anterior realiza el suministro 
de tapas que posteriormente serán montadas en el conjunto preparado en 
el palet. Sin embargo, tras esta fase resulta necesario realizar la carga de 
la tapa sobre el plato divisor. 

Para ello se ha dispuesto el manipulador de la imagen, compuesto por un cilindro 
rotolineal, encargado de realizar la elevación y posterior giro de un brazo con una pinza 
de dos dedos de apertura paralela. El giro de 180º realizado por este elemento, sitúa 
la pinza sobre el punto exacto de descarga de la tapa en la primera estación del plato 
divisor.

ESTACIÓN DE INSERCIÓN TAPA - Manual de usuario #33/29
Al igual que sucedía en la estación de inserción de eje, la última de las estaciones está encargada 
del montaje de la tapa sobre el conjunto retenido en la cinta transportadora.

Como puede observarse en la imagen, el manipulador previsto para realizar esta tarea 
presenta idénticas características que el utilizado para depositar la tapa sobre el plato divisor. 
Dispone de una pinza de apertura paralela para sujetar la tapa, que es elevada y desplazada 
realizando un giro hasta el punto de descarga mediante un actuador neumático rotolineal. *)

VAR_INPUT
	Mover			:BOOL;
END_VAR

VAR_OUTPUT
	fbController	: L2_PickAndPlace_SFC:=(dr:=dr); 
	h0 				: L1_Sensor := (uiValue:= TRUE);
	h1 				: L1_Sensor := (uiValue:= TRUE);
	v1 				: L1_Sensor := (uiValue:= TRUE);
	v0 				: L1_Sensor := (uiValue:=TRUE);
	HOR 			: L1_Actuator;
	VER 			: L1_Actuator;
	PIN 			: L1_Actuator;
	//_TapaMovida		: BOOL;
	Position		: REAL:= 0;	
END_VAR

VAR CONSTANT
	
END_VAR

METHOD ProcessCycle : BOOL
VAR_INPUT
	dr			: REFERENCE TO L1_Director;
	tapas		: REFERENCE TO L6_Tapas;	
END_VAR
IF dr.gmModeActual = L1_GEMMA.A6Inicializando THEN
	;//_TapaMovida	 				:= FALSE;
ELSE
	// Sensores y condiciones iniciales
	h0.ProcessCycle(LocalHost:=dr.gmLocalHost, sfcValue=>fbController.h0);
	h1.ProcessCycle(LocalHost:=dr.gmLocalHost, sfcValue=>fbController.h1);
	v0.ProcessCycle(LocalHost:=dr.gmLocalHost, sfcValue=>fbController.v0);
	v1.ProcessCycle(LocalHost:=dr.gmLocalHost, sfcValue=>fbController.v1);
	IC := v0.uiValue AND h0.uiValue; // el brazo está en condiciones iniciales cuando está arriba y retraído

	// Controlador
	fbController.ProcessCycle(dr.gmModeActual);
	fbController(Mover := Mover,
		dr:=dr, IC:=IC, Execute:=Execute, Ack:=Ack, Ready=>Ready, Done=>Done);
		
	// Actuadores y actualización de tapas		
	IF Ready AND Mover THEN // NOT _TapaMovida THEN 
		tapas.MoverPickAndPlace(Name:=Name, Delta:=0);// 	Position := 0;												// Inicialmente la posición es arriba
	ELSIF Done AND NOT fbController.Performed AND Mover THEN
		fbController.Performed	:= TRUE;
		//_TapaMovida				:= TRUE;
		tapas.MoverPickAndPlace(Name:=Name, Delta:=MoverMax); // //Position				:= MaxPosition;
		tapas.PostPickAndPlace(Name:=Name);  // actualizar las tapas según el nombre de brazo sea "Carga" o "Descarga"
		//IF Name='Carga' THEN
		//	tapas.PostCarga();
		//ELSE // descarga
		//	tapas.PostDesca();
		//END_IF
	ELSIF fbController.Executing AND Mover THEN // position < MaxPosition AND 
		tapas.MoverPickAndPlace(Name:=Name, Delta:=1); //Position				:= Position+1;				
	END_IF
	HOR.ProcessCycle(gmMode:=dr.gmModeActual, sfcValue:=fbController.HOR);
	VER.ProcessCycle(gmMode:=dr.gmModeActual, sfcValue:=fbController.VER);
	PIN.ProcessCycle(gmMode:=dr.gmModeActual, sfcValue:=fbController.PIN);
END_IF
END_METHOD

END_FUNCTION_BLOCK

// ---- L3 Modules/L3_PlatoDivisor.TcPOU
FUNCTION_BLOCK L3_PlatoDivisor EXTENDS L1_ModuleBase

VAR_OUTPUT	
	fbController	: L2_PlatoDivisor_SFC:=(dr:=dr);  
	d0 				: L1_Sensor := (uiValue:= TRUE);
    D_1       		: L1_Actuator;
    E_1       		: L1_Actuator;
	NumGiros 		: DINT := 0;
	Angulo			: REAL := 0;
END_VAR

VAR
	AnguloAnim		: REAL := 0;
END_VAR

METHOD ProcessCycle : BOOL 

VAR_INPUT
	dr			: REFERENCE TO L1_Director;
	tapas		: REFERENCE TO L6_Tapas;	
END_VAR
IF dr.gmModeActual = L1_GEMMA.A6Inicializando THEN
	NumGiros := 0;
	Angulo	 := 0; // -45.0;
ELSE
	// Sensores y condiciones iniciales
	d0.ProcessCycle(LocalHost:=dr.gmLocalHost, sfcValue=>fbController.d0);
	IC := d0.uiValue;
	
	// Controlador
	fbController.ProcessCycle(dr.gmModeActual);
	fbController(
		dr:=dr, IC:=IC, Execute:=Execute, Ack:=Ack, Ready=>Ready, Done=>Done);
	IF fbController.Done AND NOT fbController.Performed THEN
		fbController.Performed 	:= TRUE;
		NumGiros 				:= NumGiros + 1;
		AnguloAnim				:= 0;		
	ELSIF fbController.Executing AND anguloanim >-35.0 THEN  
		AnguloAnim 	:= anguloanim - 0.2;	
	END_IF	
	Angulo 					:= AnguloAnim -45.0 * TO_REAL(NumGiros MOD 8); // 
	// Actuadores y actualización de tapas
	D_1.ProcessCycle(gmMode:=dr.gmModeActual, sfcValue:=fbController.D_1);
	E_1.ProcessCycle(gmMode:=dr.gmModeActual, sfcValue:=fbController.E_1);
END_IF
END_METHOD

END_FUNCTION_BLOCK

// ---- L4 Station Controllers/L4_FMS205_F1Producir_SFC.TcPOU
FUNCTION_BLOCK L4_FMS205_F1Producir_SFC EXTENDS L1_ControllerBase_SFC

VAR_IN_OUT
	Alime			: L3_Alimentador;
	Carga		 	: L3_PickAndPlace;
	Medid			: L3_MedidorTapa;
	Induc		 	: L3_CaptadorInductivo;
	Fotoe			: L3_DetectorFotoelectrico;
	Evacu		 	: L3_Evacuador;
	Desca			: L3_PickAndPlace;
	Plato			: L3_PlatoDivisor;
	Cinta			: L3_Cinta;
END_VAR

